METHOD setLength
  VAR
    i : UINT;
  END_VAR
                  FOR i:=0 TO cBufferSize DO
	IF (lBuffer[i] = 0) THEN
		lLength := i;
		
		IF (i>0) THEN
			lCharacters := lLength - 1;
		ELSE
			lCharacters := 0;			
		END_IF
		
		RETURN;
	END_IF
END_FOR
                
END_METHOD

METHOD appendPair
  VAR_INPUT
    parameter : STRING;
    value : STRING;
    quoted : BOOL;
    comma : BOOL;
  END_VAR
  VAR
    stmp : STRING;
  END_VAR
                  IF (comma) THEN
	stmp := CONCAT(', "',parameter);
ELSE
	stmp := CONCAT('"',parameter);
END_IF

IF (quoted) THEN
	stmp := CONCAT(stmp,'":"');
	stmp := CONCAT(stmp,value);
	stmp := CONCAT(stmp,'"');	
ELSE
	stmp := CONCAT(stmp,'":');
	stmp := CONCAT(stmp,value);
END_IF

append(stmp);
                
END_METHOD

METHOD recordTerminatorWithNewline
                  recordTerminator();
newline();
                
END_METHOD

PROPERTY Buffer : POINTER TO BYTE
GET
                    Buffer := ADR(lBuffer[0]);
                  
END_GET
END_PROPERTY

PROPERTY CurrentToken : t_parse_token_type
GET
                    CurrentToken := lCurrentToken;
                  
END_GET
END_PROPERTY

PROPERTY Length : UINT
GET
                    Length := lLength;
                  
END_GET
SET
                    lLength := Length;
checkTermination();

                  
END_SET
END_PROPERTY

PROPERTY Overflow : BOOL
GET
                    Overflow := lOverflow;
                  
END_GET
END_PROPERTY

PROPERTY NewlineStr : t_short_string
GET
                    NewlineStr := lNewline;
                  
END_GET
SET
                    lNewline := NewlineStr;
                  
END_SET
END_PROPERTY

PROPERTY Characters : UINT
GET
                    Characters := lCharacters;
                  
END_GET
END_PROPERTY

PROPERTY RecordInitiatorStr : t_short_string
GET
                    RecordInitiatorStr := lRecordInitiator;
                  
END_GET
SET
                    lRecordInitiator := RecordInitiatorStr;
                  
END_SET
END_PROPERTY

PROPERTY IndentStr : t_short_string
GET
                    IndentStr := lIndentStr;
                  
END_GET
SET
                    lIndentStr := IndentStr;
                  
END_SET
END_PROPERTY

PROPERTY RecordTerminatorStr : t_short_string
GET
                    RecordTerminatorStr := lRecordTerminator;
                  
END_GET
SET
                    lRecordTerminator := RecordTerminatorStr;
                  
END_SET
END_PROPERTY

PROPERTY BufferSize : UINT
GET
                    BufferSize := cBufferSize + 1;
                  
END_GET
END_PROPERTY
END_FUNCTION_BLOCK

FUNCTION_BLOCK StringStorex EXTENDS PersistentValue
  VAR CONSTANT
    cBufferSize : UINT := 24000;
  END_VAR
  VAR
    lValue : ARRAY[0..cBufferSize] OF BYTE;
    lLength : UINT := 0;
  END_VAR

            
          

METHOD initialize
                  lData := ADR(lValue[0]);
lCount := SIZEOF(lValue);

SUPER^.initialize();


                
END_METHOD

METHOD append
                  
                
END_METHOD

METHOD clear
                  lLength := 0;
lValue[0] := 0;
                
END_METHOD
END_FUNCTION_BLOCK

FUNCTION allocateLongString : REFERENCE TO t_long_string
  VAR_INPUT
    target : REFERENCE TO t_long_string;
  END_VAR
  VAR
    ptr : POINTER TO t_long_string;
  END_VAR

            IF (__ISVALIDREF(target)) THEN
	allocateLongString REF= target;
	RETURN;
END_IF

ptr := __NEW(t_long_string);
_countLongString := _countLongString + 1;

IF (ptr=0) THEN
	gCodeErrorHandler(pMessage:='Memory allocation failed for <t_my_string>');
	allocateLongString REF= _defaultLongString;
	RETURN;
END_IF

ptr^ := concat('allocated:',UINT_TO_STRING(_countLongString));
allocateLongString REF= ptr^;

          
END_FUNCTION

FUNCTION defineOption_1
  VAR_INPUT
    option : INT;
    token : t_token_string;
    description : t_medium_string;
  END_VAR
  VAR
    ptrptr : POINTER TO POINTER TO t_enum_option_definition;
    ptr : POINTER TO t_enum_option_definition;
    index : USINT;
    lFailed : BOOL;
    lEnumOptionMax : USINT;
  END_VAR

            index := INT_TO_USINT(option);

IF ((index>lEnumOptionMax) OR
	(ptrptr=0)) THEN
	lFailed := TRUE;
	RETURN;
END_IF

IF (ptrptr[index]=0) THEN
	gCodeErrorHandler(pMessage:='EnumRegister option already registered - check for duplicates');
	lFailed := TRUE;
	RETURN;
END_IF

ptr := __NEW(t_enum_option_definition);

IF (ptr=0) THEN
	gCodeErrorHandler(pMessage:='Memory allocation failed for enum option in <TypeHandlerEnum>');
	lFailed := TRUE;
	RETURN;
END_IF

ptrptr[index] := ptr;

ptrptr[index]^.option := option;
ptrptr[index]^.token := token;
ptrptr[index]^.description := description;
          
END_FUNCTION

FUNCTION_BLOCK TypeHandlerEnumActiveState EXTENDS TypeHandlerEnum

            
          

METHOD initialize
                  defineOption(cActiveStateNone,'none','');
defineOption(cActiveStatePre,'pre','');
defineOption(cActiveStatePost,'post','');
defineOption(cActiveStateActive,'active','');

                
END_METHOD

METHOD FB_Init : BOOL
  VAR_INPUT
    bInitRetains : BOOL;
    bInCopyCode : BOOL;
  END_VAR
                  lDefinition.option := cEnumTypeActiveState;
lDefinition.token := 'active_state';
lDefinition.description := 'States in the Active state machine';

                
END_METHOD
END_FUNCTION_BLOCK

FUNCTION_BLOCK TypeHandlerEnumBMSChargeState EXTENDS TypeHandlerEnum

            
          

METHOD initialize
                  IF ((lInitialized) OR
	(lFailed)) THEN
	RETURN;
END_IF

lEnumOptions := __NEW(ARRAY[0..cBMSChargeStateOther] OF POINTER TO t_enum_option_definition);

IF (lEnumOptions=0) THEN
	gCodeErrorHandler(pMessage:='Memory allocation failed for <TypeHandlerEnum>');
	lFailed := TRUE;
	RETURN;
END_IF

lEnumOptionMax := INT_TO_USINT(cBMSChargeStateOther);

defineOption(cBMSChargeStateShutdown,'shutdown','');
defineOption(cBMSChargeStateDC,'dc','');
defineOption(cBMSChargeStateAC,'ac','');
defineOption(cBMSChargeStateOther,'other','');

IF (NOT(lFailed)) THEN
	lInitialized := TRUE;
END_IF

                
END_METHOD

METHOD FB_Init : BOOL
  VAR_INPUT
    bInitRetains : BOOL;
    bInCopyCode : BOOL;
  END_VAR
                  lDefinition.option := cEnumTypeBMSChargeState;
lDefinition.token := 'bms_charge_state';
lDefinition.description := 'States in the BMS charge state machine';

                
END_METHOD
END_FUNCTION_BLOCK

FUNCTION_BLOCK TypeHandlerEnumBMSFaultLevel EXTENDS TypeHandlerEnum

            
          

METHOD initialize
                  IF ((lInitialized) OR
	(lFailed)) THEN
	RETURN;
END_IF

lEnumOptions := __NEW(ARRAY[0..cBMSFaultLevelSevere] OF POINTER TO t_enum_option_definition);

IF (lEnumOptions=0) THEN
	gCodeErrorHandler(pMessage:='Memory allocation failed for <TypeHandlerEnum>');
	lFailed := TRUE;
	RETURN;
END_IF

lEnumOptionMax := INT_TO_USINT(cBMSFaultLevelSevere);

defineOption(cBMSFaultLevelNone,'none','');
defineOption(cBMSFaultLevelLow,'low','');
defineOption(cBMSFaultLevelMedium,'medium','');
defineOption(cBMSFaultLevelSevere,'severe','');

IF (NOT(lFailed)) THEN
	lInitialized := TRUE;
END_IF

                
END_METHOD

METHOD FB_Init : BOOL
  VAR_INPUT
    bInitRetains : BOOL;
    bInCopyCode : BOOL;
  END_VAR
                  lDefinition.option := cEnumTypeBMSFaultLevel;
lDefinition.token := 'bms_fault_level';
lDefinition.description := 'BMS fault level';

                
END_METHOD
END_FUNCTION_BLOCK

FUNCTION_BLOCK TypeHandlerEnumBMSState EXTENDS TypeHandlerEnum

            
          

METHOD initialize
                  IF ((lInitialized) OR
	(lFailed)) THEN
	RETURN;
END_IF

lEnumOptions := __NEW(ARRAY[0..cBMSStateConnected] OF POINTER TO t_enum_option_definition);

IF (lEnumOptions=0) THEN
	gCodeErrorHandler(pMessage:='Memory allocation failed for <TypeHandlerEnum>');
	lFailed := TRUE;
	RETURN;
END_IF

lEnumOptionMax := INT_TO_USINT(cBMSStateConnected);

defineOption(cBMSStateShutdown,'shutdown','');
defineOption(cBMSStateStandby,'standby','');
defineOption(cBMSStateDisconnected,'disconnected','');
defineOption(cBMSStateConnected,'connected','');

IF (NOT(lFailed)) THEN
	lInitialized := TRUE;
END_IF

                
END_METHOD

METHOD FB_Init : BOOL
  VAR_INPUT
    bInitRetains : BOOL;
    bInCopyCode : BOOL;
  END_VAR
                  lDefinition.option := cEnumTypeBMSState;
lDefinition.token := 'bms_state';
lDefinition.description := 'States in the BMS state machine';

                
END_METHOD
END_FUNCTION_BLOCK

FUNCTION_BLOCK TypeHandlerEnumChannelMask EXTENDS TypeHandlerEnum

            
          

METHOD initialize
                  IF ((lInitialized) OR
	(lFailed)) THEN
	RETURN;
END_IF

lEnumOptions := __NEW(ARRAY[0..9] OF POINTER TO t_enum_option_definition);

IF (lEnumOptions=0) THEN
	gCodeErrorHandler(pMessage:='Memory allocation failed for <TypeHandlerEnum>');
	lFailed := TRUE;
	RETURN;
END_IF

lEnumOptionMax := INT_TO_USINT(mapping(cChannelEdgeTrace));

defineOption(cChannelNone,'none','');
defineOption(cChannelUIRadio,'Radio','');
defineOption(cChannelUICabin,'Cabin','');
defineOption(cChannelLogTCP,'Log','');
defineOption(cChannelUIRCache,'UIRCache','');
defineOption(cChannelMaster,'Master','');
defineOption(cChannelEdgeLog,'EdgeLog','');
defineOption(cChannelEdgeStateMetric,'EdgeStateMetric','');
defineOption(cChannelEdgeValueMetric,'EdgeValueMetric','');
defineOption(cChannelEdgeTrace,'EdgeTrace','');
	
IF (NOT(lFailed)) THEN
	lInitialized := TRUE;
END_IF

                
END_METHOD

METHOD FB_Init : BOOL
  VAR_INPUT
    bInitRetains : BOOL;
    bInCopyCode : BOOL;
  END_VAR
                  lDefinition.option := cEnumTypeChannelMask;
lDefinition.token := 'channel_id';
lDefinition.description := 'Channel identifiers (mask)';


                
END_METHOD

METHOD mapping : USINT
  VAR_INPUT
    option : INT;
  END_VAR
                  mapping := 0;

CASE option OF
	cChannelNone:
		mapping := 0;

	cChannelUIRadio:
		mapping := 1;

	cChannelUICabin:
		mapping := 2;

	cChannelLogTCP:
		mapping := 3;

	cChannelUIRCache:
		mapping := 4;

	cChannelMaster:
		mapping := 5;
		
	cChannelEdgeLog:
		mapping := 6;

	cChannelEdgeStateMetric:
		mapping := 7;

	cChannelEdgeValueMetric:
		mapping := 8;

	cChannelEdgeTrace:
		mapping := 9;
END_CASE
	
                
END_METHOD
END_FUNCTION_BLOCK

FUNCTION_BLOCK TypeHandlerEnumChargeQualifier EXTENDS TypeHandlerEnum

            
          

METHOD initialize
                  IF ((lInitialized) OR
	(lFailed)) THEN
	RETURN;
END_IF

lEnumOptions := __NEW(ARRAY[0..cChargeQualifierNone] OF POINTER TO t_enum_option_definition);

IF (lEnumOptions=0) THEN
	gCodeErrorHandler(pMessage:='Memory allocation failed for <TypeHandlerEnum>');
	lFailed := TRUE;
	RETURN;
END_IF

lEnumOptionMax := INT_TO_USINT(cChargeQualifierNone);

defineOption(cChargeQualifierBoth,'both','');
defineOption(cChargeQualifierCharge,'charge','');
defineOption(cChargeQualifierDischarge,'discharge','');
defineOption(cChargeQualifierNone,'none','');

IF (NOT(lFailed)) THEN
	lInitialized := TRUE;
END_IF

                
END_METHOD

METHOD FB_Init : BOOL
  VAR_INPUT
    bInitRetains : BOOL;
    bInCopyCode : BOOL;
  END_VAR
                  lDefinition.option := cEnumTypeChargeQualifier;
lDefinition.token := 'charge_qualifier';
lDefinition.description := 'Charge modulation qualifier options';

                
END_METHOD
END_FUNCTION_BLOCK

FUNCTION_BLOCK TypeHandlerEnumDataType EXTENDS TypeHandlerEnum

            
          

METHOD initialize
                  IF ((lInitialized) OR
	(lFailed)) THEN
	RETURN;
END_IF

lEnumOptions := __NEW(ARRAY[0..cDataTypeBool] OF POINTER TO t_enum_option_definition);

IF (lEnumOptions=0) THEN
	gCodeErrorHandler(pMessage:='Memory allocation failed for <TypeHandlerEnum>');
	lFailed := TRUE;
	RETURN;
END_IF

lEnumOptionMax := INT_TO_USINT(cDataTypeBool);
	
defineOption(cDataTypeNone,'none','');
defineOption(cDataTypeEnum,'enum','');
defineOption(cDataTypeString,'string','');
defineOption(cDataTypeUSINT,'usint','');
defineOption(cDataTypeUINT,'uint','');
defineOption(cDataTypeULINT,'ulint','');
defineOption(cDataTypeUDINT,'udint','');
defineOption(cDataTypeINT,'int','');
defineOption(cDataTypePercentage,'percentage','');
defineOption(cDataTypeReal,'real','');
defineOption(cDataTypeDWORD,'dword','');
defineOption(cDataTypeBool,'bool','');

IF (NOT(lFailed)) THEN
	lInitialized := TRUE;
END_IF

                
END_METHOD

METHOD FB_Init : BOOL
  VAR_INPUT
    bInitRetains : BOOL;
    bInCopyCode : BOOL;
  END_VAR
                  lDefinition.option := cEnumTypeDataType;
lDefinition.token := 'data_type';
lDefinition.description := 'Native data types';

                
END_METHOD
END_FUNCTION_BLOCK

FUNCTION_BLOCK TypeHandlerEnumDebugMask EXTENDS TypeHandlerEnum

            
          

METHOD initialize
                  IF ((lInitialized) OR
	(lFailed)) THEN
	RETURN;
END_IF

lEnumOptions := __NEW(ARRAY[0..7] OF POINTER TO t_enum_option_definition);

IF (lEnumOptions=0) THEN
	gCodeErrorHandler(pMessage:='Memory allocation failed for <TypeHandlerEnum>');
	lFailed := TRUE;
	RETURN;
END_IF

lEnumOptionMax := INT_TO_USINT(mapping(cDebugSimulateC));

defineOption(cDebugNone,'none','');
defineOption(cDebugWaitForLog,'wait_for_log','');
defineOption(cDebugEnableFailSafeOnCrash,'enbl_fail_safe','');
defineOption(cDebugDisableWatchdog,'dsbl_watch_dog','');
defineOption(cDebugSimulateCrash,'simulate_crash','');
defineOption(cDebugSimulateA,'simulate_a','');
defineOption(cDebugSimulateB,'simulate_b','');
defineOption(cDebugSimulateC,'simulate_c','');

IF (NOT(lFailed)) THEN
	lInitialized := TRUE;
END_IF

                
END_METHOD

METHOD FB_Init : BOOL
  VAR_INPUT
    bInitRetains : BOOL;
    bInCopyCode : BOOL;
  END_VAR
                  lDefinition.option := cEnumTypeDebugMask;
lDefinition.token := 'debug_flag';
lDefinition.description := 'Debug flag (mask)';

                
END_METHOD

METHOD mapping : USINT
  VAR_INPUT
    option : INT;
  END_VAR
                  mapping := 0;

CASE option OF
	cDebugNone:
		mapping := 0;

	cDebugWaitForLog:
		mapping := 1;

	cDebugEnableFailSafeOnCrash:
		mapping := 2;

	cDebugDisableWatchdog:
		mapping := 3;

	cDebugSimulateCrash:
		mapping := 4;

	cDebugSimulateA:
		mapping := 5;

	cDebugSimulateB:
		mapping := 6;

	cDebugSimulateC:
		mapping := 7;
END_CASE

	
                
END_METHOD
END_FUNCTION_BLOCK

FUNCTION_BLOCK TypeHandlerEnumExecuteReturn EXTENDS TypeHandlerEnum

            
          

METHOD initialize
                  IF ((lInitialized) OR
	(lFailed)) THEN
	RETURN;
END_IF

lEnumOptions := __NEW(ARRAY[0..cExecuteReturnReadOnly] OF POINTER TO t_enum_option_definition);

IF (lEnumOptions=0) THEN
	gCodeErrorHandler(pMessage:='Memory allocation failed for <TypeHandlerEnum>');
	lFailed := TRUE;
	RETURN;
END_IF

lEnumOptionMax := INT_TO_USINT(cExecuteReturnReadOnly);

defineOption(cExecuteReturnOK,'OK','');
defineOption(cExecuteReturnUnknownArgumentValue,'bad_arg_value','');
defineOption(cExecuteReturnUnsupportedForParticleType,'bad_for_context','');
defineOption(cExecuteReturnNullParticle,'null_object','');
defineOption(cExecuteReturnSetOverflow,'set_overflow','');
defineOption(cExecuteReturnUnknownOption,'bad_option','');	
defineOption(cExecuteReturnOKNOK,'returned_NOK','');
defineOption(cExecuteReturnUnknownCommand,'bad_command','');
defineOption(cExecuteReturnUnknownParameter,'bad_parameter','');
defineOption(cExecuteReturnUnsupportedRecurse,'illegal_recurse','');
defineOption(cExecuteReturnExecutionQueueOverflow,'queue_overflow','');
defineOption(cExecuteReturnExecutionQueueNullParticle,'null_queue_obj','');
defineOption(cExecuteReturnParseParameterError,'parameter_syntax','');
defineOption(cExecuteReturnUnknownOptionChannelMask,'bad_channel','');
defineOption(cExecuteReturnUnknownOptionDebugMask,'bad_debug_flag','');
defineOption(cExecuteReturnIllegalIndex,'illegal_index','');
defineOption(cExecuteReturnMissingArgument,'missing_arg','');
defineOption(cExecuteReturnTooFewArguments,'missing_args','');
defineOption(cExecuteReturnTooManyArguments,'extra_args','');
defineOption(cExecuteReturnInternalError,'internal','');
defineOption(cExecuteReturnPersistFailed,'persist_failed','');
defineOption(cExecuteReturnUnprocessedArguments,'unproc_args','');
defineOption(cExecuteReturnExecutionExecutorFailed,'monitor_failed','');
defineOption(cExecuteReturnExecutionSyntax,'syntax_error','');
defineOption(cExecuteReturnReadOnly,'read_only','');

IF (NOT(lFailed)) THEN
	lInitialized := TRUE;
END_IF

                
END_METHOD

METHOD FB_Init : BOOL
  VAR_INPUT
    bInitRetains : BOOL;
    bInCopyCode : BOOL;
  END_VAR
                  lDefinition.option := cEnumTypeExecuteReturn;
lDefinition.token := 'execute_return';
lDefinition.description := 'Execution exit codes';

                
END_METHOD
END_FUNCTION_BLOCK

FUNCTION_BLOCK TypeHandlerEnumFunctionalMode EXTENDS TypeHandlerEnum

            
          

METHOD initialize
                  IF ((lInitialized) OR
	(lFailed)) THEN
	RETURN;
END_IF

lEnumOptions := __NEW(ARRAY[0..cFunctionalModeTopbeamConfiguration] OF POINTER TO t_enum_option_definition);

IF (lEnumOptions=0) THEN
	gCodeErrorHandler(pMessage:='Memory allocation failed for <TypeHandlerEnum>');
	lFailed := TRUE;
	RETURN;
END_IF

lEnumOptionMax := INT_TO_USINT(cFunctionalModeTopbeamConfiguration);

defineOption(cFunctionalModeAny,'any','');
defineOption(cFunctionalModeDefault,'default','');
defineOption(cFunctionalModeTravel,'travel','');
defineOption(cFunctionalModeLift,'lift','');
defineOption(cFunctionalModeSpreaderConfiguration,'sprd_cnfg','');
defineOption(cFunctionalModeTopbeamConfiguration,'topbm_cnfg','');

IF (NOT(lFailed)) THEN
	lInitialized := TRUE;
END_IF

                
END_METHOD

METHOD FB_Init : BOOL
  VAR_INPUT
    bInitRetains : BOOL;
    bInCopyCode : BOOL;
  END_VAR
                  lDefinition.option := cEnumTypeFunctionalMode;
lDefinition.token := 'functional_mode';
lDefinition.description := 'Machine functional mode';

                
END_METHOD
END_FUNCTION_BLOCK

FUNCTION_BLOCK TypeHandlerEnumInputMode EXTENDS TypeHandlerEnum

            
          

METHOD initialize
                  IF ((lInitialized) OR
	(lFailed)) THEN
	RETURN;
END_IF

lEnumOptions := __NEW(ARRAY[0..cInputModeTopbeamConfiguration] OF POINTER TO t_enum_option_definition);

IF (lEnumOptions=0) THEN
	gCodeErrorHandler(pMessage:='Memory allocation failed for <TypeHandlerEnum>');
	lFailed := TRUE;
	RETURN;
END_IF

lEnumOptionMax := INT_TO_USINT(cInputModeTopbeamConfiguration);

defineOption(cInputModeNone,'none','');
defineOption(cInputModeDefault,'default','');
defineOption(cInputModeSpreaderConfiguration,'sprd_cnfg','');
defineOption(cInputModeTopbeamConfiguration,'topbm_cnfg','');

IF (NOT(lFailed)) THEN
	lInitialized := TRUE;
END_IF

                
END_METHOD

METHOD FB_Init : BOOL
  VAR_INPUT
    bInitRetains : BOOL;
    bInCopyCode : BOOL;
  END_VAR
                  lDefinition.option := cEnumTypeInputMode;
lDefinition.token := 'input_mode';
lDefinition.description := 'Machine input mode';

                
END_METHOD
END_FUNCTION_BLOCK

FUNCTION_BLOCK TypeHandlerEnumLockState EXTENDS TypeHandlerEnum

            
          

METHOD initialize
                  IF ((lInitialized) OR
	(lFailed)) THEN
	RETURN;
END_IF

lEnumOptions := __NEW(ARRAY[0..cLockStatePartial] OF POINTER TO t_enum_option_definition);

IF (lEnumOptions=0) THEN
	gCodeErrorHandler(pMessage:='Memory allocation failed for <TypeHandlerEnum>');
	lFailed := TRUE;
	RETURN;
END_IF

lEnumOptionMax := INT_TO_USINT(cLockStatePartial);

defineOption(cLockStateNone,'none','');
defineOption(cLockStateUnlocked,'unlocked','');
defineOption(cLockStateLocked,'locked','');
defineOption(cLockStatePartial,'partial','');

IF (NOT(lFailed)) THEN
	lInitialized := TRUE;
END_IF

                
END_METHOD

METHOD FB_Init : BOOL
  VAR_INPUT
    bInitRetains : BOOL;
    bInCopyCode : BOOL;
  END_VAR
                  lDefinition.option := cEnumTypeLockState;
lDefinition.token := 'lock_state';
lDefinition.description := 'Twistlock lock state';

                
END_METHOD
END_FUNCTION_BLOCK

FUNCTION_BLOCK TypeHandlerEnumOBCState EXTENDS TypeHandlerEnum

            
          

METHOD initialize
                  IF ((lInitialized) OR
	(lFailed)) THEN
	RETURN;
END_IF

lEnumOptions := __NEW(ARRAY[0..cOBCStateError] OF POINTER TO t_enum_option_definition);

IF (lEnumOptions=0) THEN
	gCodeErrorHandler(pMessage:='Memory allocation failed for <TypeHandlerEnum>');
	lFailed := TRUE;
	RETURN;
END_IF

lEnumOptionMax := INT_TO_USINT(cOBCStateError);

defineOption(cOBCStateDisconnected,'disconnect','');
defineOption(cOBCStateCharging,'charging','');
defineOption(cOBCStateStandby,'standby','');
defineOption(cOBCStateError,'error','');

IF (NOT(lFailed)) THEN
	lInitialized := TRUE;
END_IF

                
END_METHOD

METHOD FB_Init : BOOL
  VAR_INPUT
    bInitRetains : BOOL;
    bInCopyCode : BOOL;
  END_VAR
                  lDefinition.option := cEnumTypeOBCState;
lDefinition.token := 'obc_state';
lDefinition.description := 'Onboard charger state';

                
END_METHOD
END_FUNCTION_BLOCK

FUNCTION_BLOCK TypeHandlerEnumOBCStatus EXTENDS TypeHandlerEnum

            
          

METHOD initialize
                  IF ((lInitialized) OR
	(lFailed)) THEN
	RETURN;
END_IF

lEnumOptions := __NEW(ARRAY[0..cOBCStatusError] OF POINTER TO t_enum_option_definition);

IF (lEnumOptions=0) THEN
	gCodeErrorHandler(pMessage:='Memory allocation failed for <TypeHandlerEnum>');
	lFailed := TRUE;
	RETURN;
END_IF

lEnumOptionMax := INT_TO_USINT(cOBCStatusError);

defineOption(cOBCStatusNone,'none','');
defineOption(cOBCStatusCharging,'charging','');
defineOption(cOBCStatusStandby,'standby','');
defineOption(cOBCStatusError,'error','');

IF (NOT(lFailed)) THEN
	lInitialized := TRUE;
END_IF

                
END_METHOD

METHOD FB_Init : BOOL
  VAR_INPUT
    bInitRetains : BOOL;
    bInCopyCode : BOOL;
  END_VAR
                  lDefinition.option := cEnumTypeOBCStatus;
lDefinition.token := 'obc_status';
lDefinition.description := 'Onboard charger status';

                
END_METHOD
END_FUNCTION_BLOCK

FUNCTION_BLOCK TypeHandlerEnumOperatingMethod EXTENDS TypeHandlerEnum

            
          

METHOD initialize
                  IF ((lInitialized) OR
	(lFailed)) THEN
	RETURN;
END_IF

lEnumOptions := __NEW(ARRAY[0..cOperatingMethodNormal] OF POINTER TO t_enum_option_definition);

IF (lEnumOptions=0) THEN
	gCodeErrorHandler(pMessage:='Memory allocation failed for <TypeHandlerEnum>');
	lFailed := TRUE;
	RETURN;
END_IF

lEnumOptionMax := INT_TO_USINT(cOperatingMethodNormal);

defineOption(cOperatingMethodNone,'none','');
defineOption(cOperatingMethodPark,'park','');
defineOption(cOperatingMethodUnpark,'unpark','');
defineOption(cOperatingMethodLock,'lock','');
defineOption(cOperatingMethodLockWithoutPark,'lock_no_park','');
defineOption(cOperatingMethodUnlock,'unlock','');
defineOption(cOperatingMethodSlow,'slow','');
defineOption(cOperatingMethodNormal,'normal','');

IF (NOT(lFailed)) THEN
	lInitialized := TRUE;
END_IF

                
END_METHOD

METHOD FB_Init : BOOL
  VAR_INPUT
    bInitRetains : BOOL;
    bInCopyCode : BOOL;
  END_VAR
                  lDefinition.option := cEnumTypeOperatingMethod;
lDefinition.token := 'operating_method';
lDefinition.description := 'Operating mode commands';

                
END_METHOD
END_FUNCTION_BLOCK

FUNCTION_BLOCK TypeHandlerEnumProgMovCode EXTENDS TypeHandlerEnum

            
          

METHOD initialize
                  IF ((lInitialized) OR
	(lFailed)) THEN
	RETURN;
END_IF

lEnumOptions := __NEW(ARRAY[0..cOBCStatusError] OF POINTER TO t_enum_option_definition);

IF (lEnumOptions=0) THEN
	gCodeErrorHandler(pMessage:='Memory allocation failed for <TypeHandlerEnum>');
	lFailed := TRUE;
	RETURN;
END_IF

lEnumOptionMax := INT_TO_USINT(cOBCStatusError);

defineOption(cProgMovCodeNone,'none','');
defineOption(cProgMovCode_Steer_0,'steer_0','');
	
IF (NOT(lFailed)) THEN
	lInitialized := TRUE;
END_IF

                
END_METHOD

METHOD FB_Init : BOOL
  VAR_INPUT
    bInitRetains : BOOL;
    bInCopyCode : BOOL;
  END_VAR
                  lDefinition.option := cEnumTypeProgMovCode;
lDefinition.token := 'progmov_code';
lDefinition.description := 'Automation code';

                
END_METHOD
END_FUNCTION_BLOCK

FUNCTION_BLOCK TypeHandlerEnumRunState EXTENDS TypeHandlerEnum

            
          

METHOD initialize
                  IF ((lInitialized) OR
	(lFailed)) THEN
	RETURN;
END_IF

lEnumOptions := __NEW(ARRAY[0..cRunStateStop] OF POINTER TO t_enum_option_definition);

IF (lEnumOptions=0) THEN
	gCodeErrorHandler(pMessage:='Memory allocation failed for <TypeHandlerEnum>');
	lFailed := TRUE;
	RETURN;
END_IF

lEnumOptionMax := INT_TO_USINT(cRunStateStop);

defineOption(cRunStateNone,'none','');
defineOption(cRunStateStart,'start','');
defineOption(cRunStateStop,'stop','');

IF (NOT(lFailed)) THEN
	lInitialized := TRUE;
END_IF

                
END_METHOD

METHOD FB_Init : BOOL
  VAR_INPUT
    bInitRetains : BOOL;
    bInCopyCode : BOOL;
  END_VAR
                  lDefinition.option := cEnumTypeRunState;
lDefinition.token := 'run_state';
lDefinition.description := 'Run state machine';

                
END_METHOD
END_FUNCTION_BLOCK

FUNCTION_BLOCK TypeHandlerEnumSeverity EXTENDS TypeHandlerEnum

            
          

METHOD initialize
                  IF ((lInitialized) OR
	(lFailed)) THEN
	RETURN;
END_IF

lEnumOptions := __NEW(ARRAY[0..cSeverityCritical] OF POINTER TO t_enum_option_definition);

IF (lEnumOptions=0) THEN
	gCodeErrorHandler(pMessage:='Memory allocation failed for <TypeHandlerEnum>');
	lFailed := TRUE;
	RETURN;
END_IF

lEnumOptionMax := INT_TO_USINT(cSeverityCritical);

defineOption(cSeverityNone,'none','');
defineOption(cSeverityWarning,'warning','');
defineOption(cSeverityError,'error','');
defineOption(cSeverityCritical,'critical','');

IF (NOT(lFailed)) THEN
	lInitialized := TRUE;
END_IF

                
END_METHOD

METHOD FB_Init : BOOL
  VAR_INPUT
    bInitRetains : BOOL;
    bInCopyCode : BOOL;
  END_VAR
                  lDefinition.option := cEnumTypeSeverity;
lDefinition.token := 'severity';
lDefinition.description := 'Severity options';

                
END_METHOD
END_FUNCTION_BLOCK

FUNCTION_BLOCK TypeHandlerEnumShutdownCode EXTENDS TypeHandlerEnum

            
          

METHOD initialize
                  IF ((lInitialized) OR
	(lFailed)) THEN
	RETURN;
END_IF

lEnumOptions := __NEW(ARRAY[0..cShutdownCodeTrapDetected] OF POINTER TO t_enum_option_definition);

IF (lEnumOptions=0) THEN
	gCodeErrorHandler(pMessage:='Memory allocation failed for <TypeHandlerEnum>');
	lFailed := TRUE;
	RETURN;
END_IF

lEnumOptionMax := INT_TO_USINT(cShutdownCodeTrapDetected);

defineOption(cShutdownCodeUnknown,'unknown','');
defineOption(cShutdownCodeIgnition,'ignition','');
defineOption(cShutdownCodeSoftware,'software','');
defineOption(cShutdownCodeSupervisor,'supervisor','');
defineOption(cShutdownCodeCrashDetected,'crash','');
defineOption(cShutdownCodeTrapDetected,'trap','');

IF (NOT(lFailed)) THEN
	lInitialized := TRUE;
END_IF

                
END_METHOD

METHOD FB_Init : BOOL
  VAR_INPUT
    bInitRetains : BOOL;
    bInCopyCode : BOOL;
  END_VAR
                  lDefinition.option := cEnumTypeShutdownCode;
lDefinition.token := 'shutdown_code';
lDefinition.description := 'Device shutdown diagnostic';

                
END_METHOD
END_FUNCTION_BLOCK

FUNCTION_BLOCK TypeHandlerEnumSteerMode EXTENDS TypeHandlerEnum

            
          

METHOD initialize
                  IF ((lInitialized) OR
	(lFailed)) THEN
	RETURN;
END_IF

lEnumOptions := __NEW(ARRAY[0..cSteerModeCustom] OF POINTER TO t_enum_option_definition);

IF (lEnumOptions=0) THEN
	gCodeErrorHandler(pMessage:='Memory allocation failed for <TypeHandlerEnum>');
	lFailed := TRUE;
	RETURN;
END_IF

lEnumOptionMax := INT_TO_USINT(cSteerModeCustom);

defineOption(cSteerModeNone,'none','');
defineOption(cSteerMode4WS,'4ws','');
defineOption(cSteerModeLateral,'lateral','');
defineOption(cSteerModeCarousel,'carousel','');
defineOption(cSteerModeReconfigure,'reconfigure','');
defineOption(cSteerModeLateralNeg90,'lat_neg_90','');
defineOption(cSteerModeLateralPos90,'lat_pos_90','');
defineOption(cSteerModeCustom,'custom','');

IF (NOT(lFailed)) THEN
	lInitialized := TRUE;
END_IF

                
END_METHOD

METHOD FB_Init : BOOL
  VAR_INPUT
    bInitRetains : BOOL;
    bInCopyCode : BOOL;
  END_VAR
                  lDefinition.option := cEnumTypeSteerMode;
lDefinition.token := 'steer_mode';
lDefinition.description := 'Steering modes';

                
END_METHOD
END_FUNCTION_BLOCK

FUNCTION_BLOCK TypeHandlerEnumSubsystem EXTENDS TypeHandlerEnum

            
          

METHOD initialize
                  IF ((lInitialized) OR
	(lFailed)) THEN
	RETURN;
END_IF

lEnumOptions := __NEW(ARRAY[0..cSubsystemMachine] OF POINTER TO t_enum_option_definition);

IF (lEnumOptions=0) THEN
	gCodeErrorHandler(pMessage:='Memory allocation failed for <TypeHandlerEnum>');
	lFailed := TRUE;
	RETURN;
END_IF

lEnumOptionMax := INT_TO_USINT(cSubsystemMachine);

defineOption(cSubsystemNone,'none','');
defineOption(cSubsystemSpreader,'Spreader','');
defineOption(cSubsystemBeacons,'Beacons','');
defineOption(cSubsystemCabin,'Cabin','');
defineOption(cSubsystemLights,'Lights','');
defineOption(cSubsystemPowerpack,'owerpack','');
defineOption(cSubsystemSideshiftAB,'SideshiftAB','');
defineOption(cSubsystemSideshiftCD,'SideshiftCD','');
defineOption(cSubsystemSpreaderPowerPack,'SprPowerPack','');
defineOption(cSubsystemSteerA,'SteerA','');
defineOption(cSubsystemSteerB,'SteerB','');
defineOption(cSubsystemSteerC,'SteerC','');
defineOption(cSubsystemSteerD,'SteerD','');
defineOption(cSubsystemTravelA,'TravelA','');
defineOption(cSubsystemTravelB,'TravelB','');
defineOption(cSubsystemTravelC,'TravelC','');
defineOption(cSubsystemTravelD,'TravelD','');
defineOption(cSubsystemWinchA,'WinchA','');
defineOption(cSubsystemWinchB,'WinchB','');
defineOption(cSubsystemWinchC,'WinchC','');
defineOption(cSubsystemWinchD,'WinchD','');
defineOption(cSubsystemTwistlockA,'TwistlockA','');
defineOption(cSubsystemTwistlockB,'TwistlockB','');
defineOption(cSubsystemTwistlockC,'TwistlockC','');
defineOption(cSubsystemTwistlockD,'TwistlockD','');
defineOption(cSubsystemTopbeamAB,'TopbeamAB','');
defineOption(cSubsystemTopbeamCD,'TopbeamCD','');
defineOption(cSubsystemCANBusSystem,'CANBusSystem','');
defineOption(cSubsystemCANBusDrive,'CANBusDrive','');
defineOption(cSubsystemBattery,'Battery','');
defineOption(cSubsystemSecondary,'Secondary','');
defineOption(cSubsystemUInterface,'UInterface','');
defineOption(cSubsystemHydraulics,'Hydraulics','');
defineOption(cSubsystemLift,'Lift','');
defineOption(cSubsystemTravel,'Travel','');
defineOption(cSubsystemSteer,'Steer','');
defineOption(cSubsystemMachine,'Machine','');

IF (NOT(lFailed)) THEN
	lInitialized := TRUE;
END_IF

                
END_METHOD

METHOD FB_Init : BOOL
  VAR_INPUT
    bInitRetains : BOOL;
    bInCopyCode : BOOL;
  END_VAR
                  lDefinition.option := cEnumTypeSubsystem;
lDefinition.token := 'subsystem';
lDefinition.description := 'Machine subsystems';

                
END_METHOD
END_FUNCTION_BLOCK

FUNCTION_BLOCK TypeHandlerEnumSystemControl EXTENDS TypeHandlerEnum

            
          

METHOD initialize
                  IF ((lInitialized) OR
	(lFailed)) THEN
	RETURN;
END_IF

lEnumOptions := __NEW(ARRAY[0..cSystemControlNone] OF POINTER TO t_enum_option_definition);

IF (lEnumOptions=0) THEN
	gCodeErrorHandler(pMessage:='Memory allocation failed for <TypeHandlerEnum>');
	lFailed := TRUE;
	RETURN;
END_IF

lEnumOptionMax := INT_TO_USINT(cSystemControlNone);

defineOption(cSystemControlReset,'reset','');
defineOption(cSystemControlEStop,'estop','');
defineOption(cSystemControlStop,'stop','');
defineOption(cSystemControlStart,'start','');
defineOption(cSystemControlNone,'none','');

IF (NOT(lFailed)) THEN
	lInitialized := TRUE;
END_IF

                
END_METHOD

METHOD FB_Init : BOOL
  VAR_INPUT
    bInitRetains : BOOL;
    bInCopyCode : BOOL;
  END_VAR
                  lDefinition.option := cEnumTypeSystemControl;
lDefinition.token := 'system_control';
lDefinition.description := 'Options for controlling system state';

                
END_METHOD
END_FUNCTION_BLOCK

FUNCTION_BLOCK TypeHandlerEnumSystemState EXTENDS TypeHandlerEnum

            
          

METHOD initialize
                  IF ((lInitialized) OR
	(lFailed)) THEN
	RETURN;
END_IF

lEnumOptions := __NEW(ARRAY[0..cSystemStateOperational] OF POINTER TO t_enum_option_definition);

IF (lEnumOptions=0) THEN
	gCodeErrorHandler(pMessage:='Memory allocation failed for <TypeHandlerEnum>');
	lFailed := TRUE;
	RETURN;
END_IF

lEnumOptionMax := INT_TO_USINT(cSystemStateOperational);

defineOption(cSystemStateNone,'none','');
defineOption(cSystemStateInitialized,'initialized','');
defineOption(cSystemStateStandby,'standby','');
defineOption(cSystemStatePreparing,'preparing','');
defineOption(cSystemStateCharging,'charging','');
defineOption(cSystemStatePreOperational,'pre_operational','');
defineOption(cSystemStatePoweringDown,'powering_down','');
defineOption(cSystemStatePoweringUp,'powering_up','');
defineOption(cSystemStateGoOperational,'go_operational','');
defineOption(cSystemStateExitOperational,'exit_operational','');
defineOption(cSystemStateOperational,'operational','');

IF (NOT(lFailed)) THEN
	lInitialized := TRUE;
END_IF

                
END_METHOD

METHOD FB_Init : BOOL
  VAR_INPUT
    bInitRetains : BOOL;
    bInCopyCode : BOOL;
  END_VAR
                  lDefinition.option := cEnumTypeSystemState;
lDefinition.token := 'system_state';
lDefinition.description := 'System state machine';

                
END_METHOD
END_FUNCTION_BLOCK

FUNCTION_BLOCK TypeHandlerEnumTMSState EXTENDS TypeHandlerEnum

            
          

METHOD initialize
                  IF ((lInitialized) OR
	(lFailed)) THEN
	RETURN;
END_IF

lEnumOptions := __NEW(ARRAY[0..cTMSStateCirculation] OF POINTER TO t_enum_option_definition);

IF (lEnumOptions=0) THEN
	gCodeErrorHandler(pMessage:='Memory allocation failed for <TypeHandlerEnum>');
	lFailed := TRUE;
	RETURN;
END_IF

lEnumOptionMax := INT_TO_USINT(cTMSStateCirculation);

defineOption(cTMSStateShutdown,'shutdown','');
defineOption(cTMSStateCooling,'cooling','');
defineOption(cTMSStateHeating,'heating','');
defineOption(cTMSStateCirculation,'circulation','');

IF (NOT(lFailed)) THEN
	lInitialized := TRUE;
END_IF

                
END_METHOD

METHOD FB_Init : BOOL
  VAR_INPUT
    bInitRetains : BOOL;
    bInCopyCode : BOOL;
  END_VAR
                  lDefinition.option := cEnumTypeTMSState;
lDefinition.token := 'tms_state';
lDefinition.description := 'Battery thermal management state';

                
END_METHOD
END_FUNCTION_BLOCK

FUNCTION_BLOCK TypeHandlerEnumTokenType EXTENDS TypeHandlerEnum

            
          

METHOD initialize
                  IF ((lInitialized) OR
	(lFailed)) THEN
	RETURN;
END_IF

lEnumOptions := __NEW(ARRAY[0..cTokenImport] OF POINTER TO t_enum_option_definition);

IF (lEnumOptions=0) THEN
	gCodeErrorHandler(pMessage:='Memory allocation failed for <TypeHandlerEnum>');
	lFailed := TRUE;
	RETURN;
END_IF

lEnumOptionMax := INT_TO_USINT(cTokenImport);

defineOption(cTokenNone,'none','');
defineOption(cTokenDescribe,'describe','');
defineOption(cTokenSyntax,'syntax','');
defineOption(cTokenVerify,'verify','');
defineOption(cTokenIdentify,'identify','');
defineOption(cTokenRegister,'register','');
defineOption(cTokenConfigure,'configure','');
defineOption(cTokenSetFailSafeMode,'failsafe_set','');
defineOption(cTokenClearFailSafeMode,'failsafe_clr','');
defineOption(cTokenFailSafeConfig,'failsafe_cnfg','');
defineOption(cTokenProceed,'proceed','');
defineOption(cTokenList,'list','');
defineOption(cTokenDebugMaskAdd,'debug_add','');
defineOption(cTokenDebugMaskDelete,'debug_del','');
defineOption(cTokenDebugMaskClear,'debug_clr','');
defineOption(cTokenClose,'close','');
defineOption(cTokenExport,'export','');
defineOption(cTokenClear,'clear','');
defineOption(cTokenDeregister,'deregister','');
defineOption(cTokenTrigger,'trigger','');
defineOption(cTokenChannelMaskAdd,'chanmask_add','');
defineOption(cTokenChannelMaskDelete,'chanmask_del','');
defineOption(cTokenChannelMaskClear,'chanmask_clr','');
defineOption(cTokenChannelIndex,'channel','');
defineOption(cTokenValue,'value','');
defineOption(cTokenOverrideValue,'override_value','');
defineOption(cTokenOverride,'override','');
defineOption(cTokenValueType,'value_type','');
defineOption(cTokenMeaning,'meaning','');
defineOption(cTokenOverrideMeaning,'override_meaning','');
defineOption(cTokenRawIndex,'raw_index','');
defineOption(cTokenIndex,'index','');
defineOption(cTokenUnknown,'unknown','');
defineOption(cTokenObject,'object','');
defineOption(cTokenFeature,'arg','');
defineOption(cTokenZero,'zero','');
defineOption(sTokenUpper,'upper','');
defineOption(cTokenImport,'import','');

IF (NOT(lFailed)) THEN
	lInitialized := TRUE;
END_IF

                
END_METHOD

METHOD FB_Init : BOOL
  VAR_INPUT
    bInitRetains : BOOL;
    bInCopyCode : BOOL;
  END_VAR
                  lDefinition.option := cEnumTypeTokenType;
lDefinition.token := 'token_type';
lDefinition.description := 'Standard tokens';

                
END_METHOD
END_FUNCTION_BLOCK

FUNCTION_BLOCK TypeHandlerEnumUIEventCode EXTENDS TypeHandlerEnum

            
          

METHOD initialize
                  IF ((lInitialized) OR
	(lFailed)) THEN
	RETURN;
END_IF

lEnumOptions := __NEW(ARRAY[0..cUIEventCodeProgMovStart] OF POINTER TO t_enum_option_definition);

IF (lEnumOptions=0) THEN
	gCodeErrorHandler(pMessage:='Memory allocation failed for <TypeHandlerEnum>');
	lFailed := TRUE;
	RETURN;
END_IF

lEnumOptionMax := INT_TO_USINT(cUIEventCodeProgMovStart);

defineOption(cUIEventCodeNone,'none','');
defineOption(cUIEventCodeToggleLights,'toggle_lights','');
defineOption(cUIEventCodeUIModeResponse,'ui_mode_resp','');
defineOption(cUIEventCodeToggleSpreaderConfiguration,'sprd_cnfg','');
defineOption(cUIEventCodeSpreaderExtensionAutoCommand,'sprd_extend','');
defineOption(cUIEventCodeSpreaderRetractionAutoCommand,'sprd_retract','');
defineOption(cUIEventCodeInitiate,'initiate','');
defineOption(cUIEventCodeStart,'start','');
defineOption(cUIEventCodeStop,'stop','');
defineOption(cUIEventCodeProgMovStart,'prog_move_start','');

IF (NOT(lFailed)) THEN
	lInitialized := TRUE;
END_IF

                
END_METHOD

METHOD FB_Init : BOOL
  VAR_INPUT
    bInitRetains : BOOL;
    bInCopyCode : BOOL;
  END_VAR
                  lDefinition.option := cEnumTypeUiEventCode;
lDefinition.token := 'ui_event_code';
lDefinition.description := 'User Interface event code';

                
END_METHOD
END_FUNCTION_BLOCK

FUNCTION_BLOCK TypeHandlerEnumUIOrientation EXTENDS TypeHandlerEnum

            
          

METHOD initialize
                  IF ((lInitialized) OR
	(lFailed)) THEN
	RETURN;
END_IF

lEnumOptions := __NEW(ARRAY[0..cUIOrientationOpposite] OF POINTER TO t_enum_option_definition);

IF (lEnumOptions=0) THEN
	gCodeErrorHandler(pMessage:='Memory allocation failed for <TypeHandlerEnum>');
	lFailed := TRUE;
	RETURN;
END_IF

lEnumOptionMax := INT_TO_USINT(cUIOrientationOpposite);

defineOption(cUIOrientationNone,'none','');
defineOption(cUIOrientationForward,'forward','');
defineOption(cUIOrientationSide,'side','');
defineOption(cUIOrientationReverse,'reverse','');
defineOption(cUIOrientationOpposite,'opposite','');

IF (NOT(lFailed)) THEN
	lInitialized := TRUE;
END_IF

                
END_METHOD

METHOD FB_Init : BOOL
  VAR_INPUT
    bInitRetains : BOOL;
    bInCopyCode : BOOL;
  END_VAR
                  lDefinition.option := cEnumTypeUiOrientation;
lDefinition.token := 'ui_orientation';
lDefinition.description := 'User Interface orientation';

                
END_METHOD
END_FUNCTION_BLOCK

FUNCTION_BLOCK TypeHandlerEnumValueStyle EXTENDS TypeHandlerEnum

            
          

METHOD initialize
                  IF ((lInitialized) OR
	(lFailed)) THEN
	RETURN;
END_IF

lEnumOptions := __NEW(ARRAY[0..cValueStyleTrigger] OF POINTER TO t_enum_option_definition);

IF (lEnumOptions=0) THEN
	gCodeErrorHandler(pMessage:='Memory allocation failed for <TypeHandlerEnum>');
	lFailed := TRUE;
	RETURN;
END_IF

lEnumOptionMax := INT_TO_USINT(cValueStyleTrigger);

defineOption(cValueStyleConfigurable,'configurable','');
defineOption(cValueStyleParameter,'parameter','');
defineOption(cValueStyleTrigger,'trigger','');

IF (NOT(lFailed)) THEN
	lInitialized := TRUE;
END_IF

                
END_METHOD

METHOD FB_Init : BOOL
  VAR_INPUT
    bInitRetains : BOOL;
    bInCopyCode : BOOL;
  END_VAR
                  lDefinition.option := cEnumTypeValueStyle;
lDefinition.token := 'value_style';
lDefinition.description := 'How a value is treated';

                
END_METHOD
END_FUNCTION_BLOCK

FUNCTION getStringForEventCode : t_medium_string
  VAR_INPUT
    code : t_event_code;
  END_VAR

            getStringForEventCode := 'event';

CASE code OF
	cECNone:
		getStringForEventCode := 'none';

	cECSystemControl:
		getStringForEventCode := 'SysStateCntrl';

	cECAllowUpState:
		getStringForEventCode := 'SysStateAllowUp';

	cECAllowDownState:
		getStringForEventCode := 'SysStateAllowDn';

	cECForceMaxState:
		getStringForEventCode := 'SysStateMax';

	cECNextState:
		getStringForEventCode := 'SysStateNext';

	cECModulation:
		getStringForEventCode := 'SysStateMod';

	cECChargeModulation:
		getStringForEventCode := 'SysStateChrgMod';

	cECMovementInputInterlock:
		getStringForEventCode := 'iMovInput';

	cECMovementChargeInterlock:
		getStringForEventCode := 'iMovChrg';

	cECSecondaryPowerModulation:
		getStringForEventCode := 'SecPwrMod';

	cECTransitionInitializedStandby:
		getStringForEventCode := 'sstInitStdby';

	cECTransitionStandbyPreparing:
		getStringForEventCode := 'sstStdbyPrep';

	cECTransitionStandbyInitialized:
		getStringForEventCode := 'sstStbyInit';

	cECTransitionPreparingPreOperational:
		getStringForEventCode := 'sstPrepPreOp';

	cECTransitionPreparingCharging:
		getStringForEventCode := 'sstPrepChrg';

	cECTransitionPreparingStandby:
		getStringForEventCode := 'sstPrepStdby';

	cECTransitionChargingPreparing:
		getStringForEventCode := 'sstChrgPrep';

	cECTransitionPreOperationalPreparing:
		getStringForEventCode := 'sstPreOpPrep';

	cECTransitionPoweringUpGoOperational:
		getStringForEventCode := 'sstPwrUpGoOp';

	cECTransitionGoOperationalOperational:
		getStringForEventCode := 'sstGoOpOper';

	cECTransitionExitOperationalPoweringDown:
		getStringForEventCode := 'sstExOpPwrDn';

	cECTransitionPoweringDownPreOperational:
		getStringForEventCode := 'sstPwrDnPreOp';
		
	cECMetric:
		getStringForEventCode := 'Metric';	
END_CASE

IF (strcmp(getStringForEventCode,'event')) THEN
	gEventCodeLastUnknown := code;
END_IF
          
END_FUNCTION

FUNCTION getStringForParseTokenType : t_medium_string
  VAR_INPUT
    token : t_parse_token_type;
  END_VAR

            getStringForParseTokenType := 'none';		

CASE token OF
	cParseTokenOverflow:
		getStringForParseTokenType := 'overflow';
		
	cParseTokenError:
		getStringForParseTokenType := 'error';

	cParseTokenSimple:
		getStringForParseTokenType := 'command';
		
	cParseTokenName:
		getStringForParseTokenType := 'name';
		
	cParseTokenParameter:
		getStringForParseTokenType := 'parameter';
		
	cParseTokenOption:
		getStringForParseTokenType := 'option';
	
	cParseTokenTerminator:
		getStringForParseTokenType := 'terminator';
		
	cParseTokenFinished:
		getStringForParseTokenType := 'finished';
END_CASE
          
END_FUNCTION

FUNCTION getStringForStateCode : t_medium_string
  VAR_INPUT
    code : t_state_code;
  END_VAR

            getStringForStateCode :='state';

CASE code OF
	cSCNone:
		getStringForStateCode := 'none';

	cACSteerALargeSensorDelta:
		getStringForStateCode := 'LrgSensorDelta';

	cACSecondaryNotRunning:
		getStringForStateCode := 'SecPwrNotRun';

	cACSecondaryNotRunningModulation:
		getStringForStateCode := 'SecPwrNotRunMod';

	cACSecondaryWaiting:
		getStringForStateCode := 'SecPwrWait';

	cACSecondaryRunStateMismatch:
		getStringForStateCode := 'SecPwrMismatch';

	cACSecondaryTemperature:
		getStringForStateCode := 'SecPwrTemp';
	
	cACChannelNotGood:
		getStringForStateCode := 'MasterNotGood';

	cACChannelOperationalFail:
		getStringForStateCode := 'MasterOpFail';

	cACChannelNotOperational:
		getStringForStateCode := 'MasterNotOp';

	cACChannelOverflow:
		getStringForStateCode := 'MasterOverflow';

	cACChannelSlaveFailed:
		getStringForStateCode := 'MasterSlaveFail';

	cACCANOpenSlaveNotOperational:
		getStringForStateCode := 'SlaveNotOp';

	cACCANOpenSlaveModulation:
		getStringForStateCode := 'SlaveMod';

	cACCANOpenSlaveAllowableUp:
		getStringForStateCode := 'SlaveAllowUp';

	cACCANOpenMasterNotOperational:
		getStringForStateCode := 'MasterNotOp';

	cACCANOpenMasterModulation:
		getStringForStateCode := 'MasterMod';

	cACCANOpenMasterAllowableUp:
		getStringForStateCode := 'MasterAllowUp';
	
	cACCANOpenSlaveNoValidTransmissions:
		getStringForStateCode := 'SlaveNoVldTrnms';

	cACCANOpenSlaveNotify:
		getStringForStateCode := 'SlaveNotify';

	cACCANOpenSlaveBlock:
		getStringForStateCode := 'SlaveBlock';

	cACCANOpenSlaveStop:
		getStringForStateCode := 'SlaveStop';
		
	cACUInterfaceEstop:
		getStringForStateCode := 'UIEstop';

	cACUInterfaceStop:
		getStringForStateCode := 'UIStop';

	cACUInterfaceEmgy:
		getStringForStateCode := 'UIEmgy';

	cACUInterfaceNotReady:
		getStringForStateCode := 'UINotRdy';

	cACControllerTemperatureCutback:
		getStringForStateCode := 'CntTempCutb';
		
	cACMotorTemperatureCutback:
		getStringForStateCode := 'MotTempCutb';

	cACMotorTemperatureSensor:
		getStringForStateCode := 'MotTempSensor';

	cACCoolantReservoir:
		getStringForStateCode := 'ClntReserv';

	cACCoolantTempHotCutback:
		getStringForStateCode := 'ClntTempHotCutb';

	cACCoolantTempColdCutback:
		getStringForStateCode := 'ClntTempColdCutb';

	cACCoolantHeating:
		getStringForStateCode := 'ClntHeating';

	cACCoolantChilling:
		getStringForStateCode := 'ClntChilling';

	cACCoolantSecondaryPowerFailHeatingCooling:
		getStringForStateCode := 'ClntSecFailHC';

	cACCoolantSecondaryPowerFailPump:
		getStringForStateCode := 'ClntSecFailPmp';

	cACChargerOBCError:
		getStringForStateCode := 'ChrgOBCErr';

	cACBMSAvailabilityInsufficient:
		getStringForStateCode := 'BMSAvailInsuff';

	cACBMSAvailabilityLimited:
		getStringForStateCode := 'BMSAvailLmtd';

	cBMSChargeAvailabilityLimited:
		getStringForStateCode := 'BMSChrgAvailLm';

	cBMSChargeAvailabilityLimitedSevere:
		getStringForStateCode := 'BMSChrgAvailLmSv';

	cBMSDischargeAvailabilityLimited:
		getStringForStateCode := 'BMSDschAvailLm';

	cBMSDischargeAvailabilityLimitedSevere:
		getStringForStateCode := 'BMSDschAvailLmSv';
		
	cACBMSRequestDisconnect:
		getStringForStateCode := 'BMSReqDisconnect';
	
	cACSOCBelowOperatingMinimum:
		getStringForStateCode := 'SOCLowOpMin';

	cACSOCBelowStandbyMinimum:
		getStringForStateCode := 'SOCLowStdbyMin';

	cACSOCWarningLow:
		getStringForStateCode := 'SOCWarnLow';
	
	cACBMSNotConnected:
		getStringForStateCode := 'BMSNotConnect';
		
	cACBMSFailToConnect:
		getStringForStateCode := 'BMSNotConnect';

	cACBMSChargeCutback:
		getStringForStateCode := 'BMSChrgCutb';

	cACBMSDischargeCutback:
		getStringForStateCode := 'BMSDischCutb';

	cACBackupBatteryVoltageLow:
		getStringForStateCode := 'BckupBatVltLow';

	cACBeaconsSecondaryPowerFail:
		getStringForStateCode := 'BcnsSecPwrFail';

	cACSecondaryPowerFail:
		getStringForStateCode := 'BeepSecPwrFail';

	cACTMSStateMismatch:
		getStringForStateCode := 'TMSMismatch';

	cACBMSChargeStateMismatch:
		getStringForStateCode := 'BMSChrgMismatch';
		
	cACBMSSOCMismatch:
		getStringForStateCode := 'BMSSOCMismatch';

	cACBMSVoltageMismatch:
		getStringForStateCode := 'BMSVoltMismatch';

	cACBMSCurrentMismatch:
		getStringForStateCode := 'BMSCurrMismatch';

	cACSensorRangeError:
		getStringForStateCode := 'SensorRange';

	cACHydraulicFilter:
		getStringForStateCode := 'HydFilter';

	cACHydraulicTemperature:
		getStringForStateCode := 'HydTemp';
	
	cACBrakeLowHydraulicPressure:
		getStringForStateCode := 'BrakeHydPress';

	cACOutputFailure:
		getStringForStateCode := 'OutputFailure';
	
	cACDeviceTemperature:
		getStringForStateCode := 'DeviceTemp';

	cACDeviceVoltage:
		getStringForStateCode := 'DeviceVoltage';
		
	cACSoftwareCrash:
		getStringForStateCode := 'SoftwareCrash';

	cACFailSafeMode:
		getStringForStateCode := 'FailSafeMode';
	
	cACMaintenanceMode:
		getStringForStateCode := 'MaintenanceMode';

	cACWatchdogDisabled:
		getStringForStateCode := 'WatchdogDsbld';
		
	cACExecutionFailed:
		getStringForStateCode := 'ExecutionFail';

	cACPersistedCommands:
		getStringForStateCode := 'PersistCmds';
	
	cACSoftware:
		getStringForStateCode := 'Software';

	cACConfiguration:
		getStringForStateCode := 'Configuration';

	cACVoltage:
		getStringForStateCode := 'Voltage';

	cACTemperature:
		getStringForStateCode := 'Temperature';

	cACRelayFuse:
		getStringForStateCode := 'RelayOrFuse';

	cACFuse:
		getStringForStateCode := 'Fuse';

	cACSubsystem:
		getStringForStateCode := 'Subsystem';

	cACConsumable:
		getStringForStateCode := 'Consumable';

	cACHeartbeat:
		getStringForStateCode := 'Heartbeat';

	cACOutput:
		getStringForStateCode := 'Output';

	cACControlSignal:
		getStringForStateCode := 'ControlSignal';
	
	cDCChargerStandby:
		getStringForStateCode := 'ChrgStdby';

	cDCChargerConnected:
		getStringForStateCode := 'ChrgConn';

	cDCChargerDisconnected:
		getStringForStateCode := 'ChrgDiscon';

	cDCTMSCooling:
		getStringForStateCode := 'TMSCooling';

	cDCTMSHeating:
		getStringForStateCode := 'TMSHeating';

	cDCBMSTMSCooling:
		getStringForStateCode := 'BMSTMSCooling';

	cDCBMSTMSHeating:
		getStringForStateCode := 'BMSTMSHeating';

	cDCBMSTMSNoCirculation:
		getStringForStateCode := 'BMSTMSNoCirc';

	cCCChargerStandby:
		getStringForStateCode := 'ChrgStdby';

	cCCChargerConnected:
		getStringForStateCode := 'ChrgConn';

	cCCChargerDisconnected:
		getStringForStateCode := 'ChrgDiscon';

	cCCWaitingForBrakeDisengaged:
		getStringForStateCode := 'WaitBrkDiseng';

	cCCWaitingForParked:
		getStringForStateCode := 'WaitParked';

	cCCCommandStart:
		getStringForStateCode := 'CmdStart';

	cCCCommandStop:
		getStringForStateCode := 'CmdStop';

	cCCStopOnTimeout:
		getStringForStateCode := 'StopOnTimeout';

	cCCLockoutInterlock:
		getStringForStateCode := 'iLockout';

	cCCPosOnlyInterlock:
		getStringForStateCode := 'iPosOnly';

	cCCScaledInterlock:
		getStringForStateCode := 'iScaled';

	cCCThresholdInterlock:
		getStringForStateCode := 'iThreshold';

	cCCSynchronousInterlock:
		getStringForStateCode := 'iSync';

	cCCTwistlocksReadyInterlock:
		getStringForStateCode := 'iTwistRdy';
		
	cCCAutomaticStart:
		getStringForStateCode := 'AutoStart';
		
	cCCSyncState:
		getStringForStateCode := 'SyncState';
		
	cCCCurrentUserNotEnabled:
		getStringForStateCode := 'UserDisabled';
		
	cCCStandby:
		getStringForStateCode := 'Standby';
		
	cCCCycleOutput:
		getStringForStateCode := 'CycleOutput';
END_CASE

IF (strcmp(getStringForStateCode,'state')) THEN
	gStateCodeLastUnknown := code;
END_IF
          
END_FUNCTION

FUNCTION_BLOCK GlobalTypeHandler
  VAR CONSTANT
    cEnumRegisterMax : USINT := ANY_TO_USINT(cEnumTypeDataType);
  END_VAR
  VAR
    lEnumRegister : ARRAY[1..cEnumRegisterMax] OF TypeHandlerEnum;
  END_VAR

            
          

METHOD initialize
  VAR
    ptr : POINTER TO TypeHandlerEnum;
  END_VAR
                  
ptr := ADR(lEnumRegister[cEnumTypeActiveState]);
ptr^.Definition.option := cEnumTypeActiveState;
ptr^.Definition.token := 'active_state';
ptr^.Definition.description := 'States in the Active state machine';
	
ptr^.defineOption(cActiveStateNone,'none','');
ptr^.defineOption(cActiveStatePre,'pre','');
ptr^.defineOption(cActiveStatePost,'post','');
ptr^.defineOption(cActiveStateActive,'active','');

ptr := ADR(lEnumRegister[cEnumTypeBMSChargeState]);
ptr^.Definition.option := cEnumTypeBMSChargeState;
ptr^.Definition.token := 'bms_charge_state';
ptr^.Definition.description := 'States in the BMS charge state machine';
	
ptr^.defineOption(cBMSChargeStateShutdown,'shutdown','');
ptr^.defineOption(cBMSChargeStateDC,'dc','');
ptr^.defineOption(cBMSChargeStateAC,'ac','');
ptr^.defineOption(cBMSChargeStateOther,'other','');

ptr := ADR(lEnumRegister[cEnumTypeBMSFaultLevel]);
ptr^.Definition.option := cEnumTypeBMSFaultLevel;
ptr^.Definition.token := 'bms_fault_level';
ptr^.Definition.description := 'BMS fault level';
	
ptr^.defineOption(cBMSFaultLevelNone,'none','');
ptr^.defineOption(cBMSFaultLevelLow,'low','');
ptr^.defineOption(cBMSFaultLevelMedium,'medium','');
ptr^.defineOption(cBMSFaultLevelSevere,'severe','');

ptr := ADR(lEnumRegister[cEnumTypeBMSState]);
ptr^.Definition.option := cEnumTypeBMSState;
ptr^.Definition.token := 'bms_state';
ptr^.Definition.description := 'States in the BMS state machine';
	
ptr^.defineOption(cBMSStateShutdown,'shutdown','');
ptr^.defineOption(cBMSStateStandby,'standby','');
ptr^.defineOption(cBMSStateDisconnected,'disconnected','');
ptr^.defineOption(cBMSStateConnected,'connected','');

ptr := ADR(lEnumRegister[cEnumTypeChannelMask]);
ptr^.Definition.option := cEnumTypeChannelMask;
ptr^.Definition.token := 'channel_id';
ptr^.Definition.description := 'Channel identifiers (mask)';
	
ptr^.defineOption(cChannelNone,'none','');
ptr^.defineOption(cChannelUIRadio,'Radio','');
ptr^.defineOption(cChannelUICabin,'Cabin','');
ptr^.defineOption(cChannelLogTCP,'Log','');
ptr^.defineOption(cChannelUIRCache,'UIRCache','');
ptr^.defineOption(cChannelMaster,'Master','');
ptr^.defineOption(cChannelEdgeLog,'EdgeLog','');
ptr^.defineOption(cChannelEdgeStateMetric,'EdgeStateMetric','');
ptr^.defineOption(cChannelEdgeValueMetric,'EdgeValueMetric','');
ptr^.defineOption(cChannelEdgeTrace,'EdgeTrace','');

ptr := ADR(lEnumRegister[cEnumTypeChargeQualifier]);
ptr^.Definition.option := cEnumTypeChargeQualifier;
ptr^.Definition.token := 'charge_qualifier';
ptr^.Definition.description := 'Charge modulation qualifier options';
	
ptr^.defineOption(cChargeQualifierBoth,'both','');
ptr^.defineOption(cChargeQualifierCharge,'charge','');
ptr^.defineOption(cChargeQualifierDischarge,'discharge','');
ptr^.defineOption(cChargeQualifierNone,'none','');

ptr := ADR(lEnumRegister[cEnumTypeDataType]);
ptr^.Definition.option := cEnumTypeDataType;
ptr^.Definition.token := 'data_type';
ptr^.Definition.description := 'Native data types';
	
ptr^.defineOption(cDataTypeNone,'none','');
ptr^.defineOption(cDataTypeEnum,'enum','');
ptr^.defineOption(cDataTypeString,'string','');
ptr^.defineOption(cDataTypeUSINT,'usint','');
ptr^.defineOption(cDataTypeUINT,'uint','');
ptr^.defineOption(cDataTypeULINT,'ulint','');
ptr^.defineOption(cDataTypeUDINT,'udint','');
ptr^.defineOption(cDataTypeINT,'int','');
ptr^.defineOption(cDataTypePercentage,'percentage','');
ptr^.defineOption(cDataTypeReal,'real','');
ptr^.defineOption(cDataTypeDWORD,'dword','');
ptr^.defineOption(cDataTypeBool,'bool','');

ptr := ADR(lEnumRegister[cEnumTypeDebugMask]);
ptr^.Definition.option := cEnumTypeDebugMask;
ptr^.Definition.token := 'debug_flag';
ptr^.Definition.description := 'Debug flag (mask)';
	
ptr^.defineOption(cDebugNone,'none','');
ptr^.defineOption(cDebugWaitForLog,'wait_for_log','');
ptr^.defineOption(cDebugEnableFailSafeOnCrash,'enbl_fail_safe','');
ptr^.defineOption(cDebugDisableWatchdog,'dsbl_watch_dog','');
ptr^.defineOption(cDebugSimulateCrash,'simulate_crash','');
ptr^.defineOption(cDebugSimulateA,'simulate_a','');
ptr^.defineOption(cDebugSimulateB,'simulate_b','');
ptr^.defineOption(cDebugSimulateC,'simulate_c','');

ptr := ADR(lEnumRegister[cEnumTypeExecuteOption]);
ptr^.Definition.option := cEnumTypeExecuteOption;
ptr^.Definition.token := 'execute_option';
ptr^.Definition.description := 'Options passed to execution calls';

ptr^.defineOption(cExecuteOptionNone,'none','');
ptr^.defineOption(cExecuteOptionRecurse,'recurse','');
ptr^.defineOption(cExecuteOptionVerbose,'verbose','');
ptr^.defineOption(cExecuteOptionParameter,'parameter','');
ptr^.defineOption(cExecuteOptionSyntax,'syntax','');
ptr^.defineOption(cExecuteOptionChildren,'children','');
ptr^.defineOption(cExecuteOptionExecutor,'executor','');
ptr^.defineOption(cExecuteOptionSubsystems,'subsystems','');
ptr^.defineOption(cExecuteOptionPersist,'persist','');
ptr^.defineOption(cExecuteOptionAll,'all','');
ptr^.defineOption(cExecuteOptionMetadata,'metadata','');

ptr := ADR(lEnumRegister[cEnumTypeExecuteReturn]);
ptr^.Definition.option := cEnumTypeExecuteReturn;
ptr^.Definition.token := 'execute_return';
ptr^.Definition.description := 'Execution exit codes';

ptr^.defineOption(cExecuteReturnOK,'OK','');
ptr^.defineOption(cExecuteReturnUnknownArgumentValue,'bad_arg_value','');
ptr^.defineOption(cExecuteReturnUnsupportedForParticleType,'bad_for_context','');
ptr^.defineOption(cExecuteReturnNullParticle,'null_object','');
ptr^.defineOption(cExecuteReturnSetOverflow,'set_overflow','');
ptr^.defineOption(cExecuteReturnUnknownOption,'bad_option','');	
ptr^.defineOption(cExecuteReturnOKNOK,'returned_NOK','');
ptr^.defineOption(cExecuteReturnUnknownCommand,'bad_command','');
ptr^.defineOption(cExecuteReturnUnknownParameter,'bad_parameter','');
ptr^.defineOption(cExecuteReturnUnsupportedRecurse,'illegal_recurse','');
ptr^.defineOption(cExecuteReturnExecutionQueueOverflow,'queue_overflow','');
ptr^.defineOption(cExecuteReturnExecutionQueueNullParticle,'null_queue_obj','');
ptr^.defineOption(cExecuteReturnParseParameterError,'parameter_syntax','');
ptr^.defineOption(cExecuteReturnUnknownOptionChannelMask,'bad_channel','');
ptr^.defineOption(cExecuteReturnUnknownOptionDebugMask,'bad_debug_flag','');
ptr^.defineOption(cExecuteReturnIllegalIndex,'illegal_index','');
ptr^.defineOption(cExecuteReturnMissingArgument,'missing_arg','');
ptr^.defineOption(cExecuteReturnTooFewArguments,'missing_args','');
ptr^.defineOption(cExecuteReturnTooManyArguments,'extra_args','');
ptr^.defineOption(cExecuteReturnInternalError,'internal','');
ptr^.defineOption(cExecuteReturnPersistFailed,'persist_failed','');
ptr^.defineOption(cExecuteReturnUnprocessedArguments,'unproc_args','');
ptr^.defineOption(cExecuteReturnExecutionExecutorFailed,'monitor_failed','');
ptr^.defineOption(cExecuteReturnExecutionSyntax,'syntax_error','');
ptr^.defineOption(cExecuteReturnExecutionSyntaxIncompleteRequest,'incmplt_reqst','');
ptr^.defineOption(cExecuteReturnExecutionSyntaxIncompleteParameter,'incmplt_prm','');
ptr^.defineOption(cExecuteReturnExecutionSyntaxIncompleteName,'incmplt_name','');
ptr^.defineOption(cExecuteReturnExecutionSyntaxTokenOverflow,'token_overflow','');
ptr^.defineOption(cExecuteReturnExecutionSyntaxStartWithName,'start_name','');
ptr^.defineOption(cExecuteReturnExecutionSyntaxCommandAfterName,'name_then_cmd','');
ptr^.defineOption(cExecuteReturnExecutionSyntaxDuplicateCommands,'duplicate_cmd','');
ptr^.defineOption(cExecuteReturnExecutionSyntaxUnkownName,'unknown_name','');
ptr^.defineOption(cExecuteReturnExecutionSyntaxUnkownNameForParameter,'unkn_name_par','');
ptr^.defineOption(cExecuteReturnExecutionSyntaxTooManyOptions,'excess_options','');
ptr^.defineOption(cExecuteReturnExecutionSyntaxUnbounded,'syntax_unbounded','');
ptr^.defineOption(cExecuteReturnReadOnly,'read_only','');

ptr := ADR(lEnumRegister[cEnumTypeFunctionalMode]);
ptr^.Definition.option := cEnumTypeFunctionalMode;
ptr^.Definition.token := 'functional_mode';
ptr^.Definition.description := 'Machine functional mode';

ptr^.defineOption(cFunctionalModeAny,'any','');
ptr^.defineOption(cFunctionalModeDefault,'default','');
ptr^.defineOption(cFunctionalModeTravel,'travel','');
ptr^.defineOption(cFunctionalModeLift,'lift','');
ptr^.defineOption(cFunctionalModeSpreaderConfiguration,'sprd_cnfg','');
ptr^.defineOption(cFunctionalModeTopbeamConfiguration,'topbm_cnfg','');

ptr := ADR(lEnumRegister[cEnumTypeInputMode]);
ptr^.Definition.option := cEnumTypeInputMode;
ptr^.Definition.token := 'input_mode';
ptr^.Definition.description := 'Machine input mode';
	
ptr^.defineOption(cInputModeNone,'none','');
ptr^.defineOption(cInputModeDefault,'default','');
ptr^.defineOption(cInputModeSpreaderConfiguration,'sprd_cnfg','');
ptr^.defineOption(cInputModeTopbeamConfiguration,'topbm_cnfg','');

ptr := ADR(lEnumRegister[cEnumTypeLockState]);
ptr^.Definition.option := cEnumTypeLockState;
ptr^.Definition.token := 'lock_state';
ptr^.Definition.description := 'Twistlock lock state';

ptr^.defineOption(cLockStateNone,'none','');
ptr^.defineOption(cLockStateUnlocked,'unlocked','');
ptr^.defineOption(cLockStateLocked,'locked','');
ptr^.defineOption(cLockStatePartial,'partial','');

ptr := ADR(lEnumRegister[cEnumTypeOBCState]);
ptr^.Definition.option := cEnumTypeOBCState;
ptr^.Definition.token := 'obc_state';
ptr^.Definition.description := 'Onboard charger state';

ptr^.defineOption(cOBCStateDisconnected,'disconnect','');
ptr^.defineOption(cOBCStateCharging,'charging','');
ptr^.defineOption(cOBCStateStandby,'standby','');
ptr^.defineOption(cOBCStateError,'error','');

ptr := ADR(lEnumRegister[cEnumTypeOBCStatus]);
ptr^.Definition.option := cEnumTypeOBCStatus;
ptr^.Definition.token := 'obc_status';
ptr^.Definition.description := 'Onboard charger status';

ptr^.defineOption(cOBCStatusNone,'none','');
ptr^.defineOption(cOBCStatusCharging,'charging','');
ptr^.defineOption(cOBCStatusStandby,'standby','');
ptr^.defineOption(cOBCStatusError,'error','');

ptr := ADR(lEnumRegister[cEnumTypeOperatingMethod]);
ptr^.Definition.option := cEnumTypeOperatingMethod;
ptr^.Definition.token := 'operating_method';
ptr^.Definition.description := 'Operating mode commands';

ptr^.defineOption(cOperatingMethodNone,'none','');
ptr^.defineOption(cOperatingMethodPark,'park','');
ptr^.defineOption(cOperatingMethodUnpark,'unpark','');
ptr^.defineOption(cOperatingMethodLock,'lock','');
ptr^.defineOption(cOperatingMethodLockWithoutPark,'lock_no_park','');
ptr^.defineOption(cOperatingMethodUnlock,'unlock','');
ptr^.defineOption(cOperatingMethodSlow,'slow','');
ptr^.defineOption(cOperatingMethodNormal,'normal','');

ptr := ADR(lEnumRegister[cEnumTypeProgMovCode]);
ptr^.Definition.option := cEnumTypeProgMovCode;
ptr^.Definition.token := 'progmov_code';
ptr^.Definition.description := 'Automation code';

ptr^.defineOption(cProgMovCodeNone,'none','');
ptr^.defineOption(cProgMovCode_Steer_0,'steer_0','');

ptr := ADR(lEnumRegister[cEnumTypeRunState]);
ptr^.Definition.option := cEnumTypeRunState;
ptr^.Definition.token := 'run_state';
ptr^.Definition.description := 'Run state machine';

ptr^.defineOption(cRunStateNone,'none','');
ptr^.defineOption(cRunStateStart,'start','');
ptr^.defineOption(cRunStateStop,'stop','');

ptr := ADR(lEnumRegister[cEnumTypeSeverity]);
ptr^.Definition.option := cEnumTypeSeverity;
ptr^.Definition.token := 'severity';
ptr^.Definition.description := 'Severity options';

ptr^.defineOption(cSeverityNone,'none','');
ptr^.defineOption(cSeverityWarning,'warning','');
ptr^.defineOption(cSeverityError,'error','');
ptr^.defineOption(cSeverityCritical,'critical','');

ptr := ADR(lEnumRegister[cEnumTypeShutdownCode]);
ptr^.Definition.option := cEnumTypeShutdownCode;
ptr^.Definition.token := 'shutdown_code';
ptr^.Definition.description := 'Device shutdown diagnostic';

ptr^.defineOption(cShutdownCodeUnknown,'unknown','');
ptr^.defineOption(cShutdownCodeIgnition,'ignition','');
ptr^.defineOption(cShutdownCodeSoftware,'software','');
ptr^.defineOption(cShutdownCodeSupervisor,'supervisor','');
ptr^.defineOption(cShutdownCodeCrashDetected,'crash','');
ptr^.defineOption(cShutdownCodeTrapDetected,'trap','');

ptr := ADR(lEnumRegister[cEnumTypeSteerMode]);
ptr^.Definition.option := cEnumTypeSteerMode;
ptr^.Definition.token := 'steer_mode';
ptr^.Definition.description := 'Steering modes';

ptr^.defineOption(cSteerModeNone,'none','');
ptr^.defineOption(cSteerMode4WS,'4ws','');
ptr^.defineOption(cSteerModeLateral,'lateral','');
ptr^.defineOption(cSteerModeCarousel,'carousel','');
ptr^.defineOption(cSteerModeReconfigure,'reconfigure','');
ptr^.defineOption(cSteerModeLateralNeg90,'lat_neg_90','');
ptr^.defineOption(cSteerModeLateralPos90,'lat_pos_90','');
ptr^.defineOption(cSteerModeCustom,'custom','');

ptr := ADR(lEnumRegister[cEnumTypeSubsystem]);
ptr^.Definition.option := cEnumTypeSubsystem;
ptr^.Definition.token := 'subsystem';
ptr^.Definition.description := 'Machine subsystems';

ptr^.defineOption(cSubsystemNone,'none','');
ptr^.defineOption(cSubsystemSpreader,'Spreader','');
ptr^.defineOption(cSubsystemBeacons,'Beacons','');
ptr^.defineOption(cSubsystemCabin,'Cabin','');
ptr^.defineOption(cSubsystemLights,'Lights','');
ptr^.defineOption(cSubsystemPowerpack,'owerpack','');
ptr^.defineOption(cSubsystemSideshiftAB,'SideshiftAB','');
ptr^.defineOption(cSubsystemSideshiftCD,'SideshiftCD','');
ptr^.defineOption(cSubsystemSpreaderPowerPack,'SprPowerPack','');
ptr^.defineOption(cSubsystemSteerA,'SteerA','');
ptr^.defineOption(cSubsystemSteerB,'SteerB','');
ptr^.defineOption(cSubsystemSteerC,'SteerC','');
ptr^.defineOption(cSubsystemSteerD,'SteerD','');
ptr^.defineOption(cSubsystemTravelA,'TravelA','');
ptr^.defineOption(cSubsystemTravelB,'TravelB','');
ptr^.defineOption(cSubsystemTravelC,'TravelC','');
ptr^.defineOption(cSubsystemTravelD,'TravelD','');
ptr^.defineOption(cSubsystemWinchA,'WinchA','');
ptr^.defineOption(cSubsystemWinchB,'WinchB','');
ptr^.defineOption(cSubsystemWinchC,'WinchC','');
ptr^.defineOption(cSubsystemWinchD,'WinchD','');
ptr^.defineOption(cSubsystemTwistlockA,'TwistlockA','');
ptr^.defineOption(cSubsystemTwistlockB,'TwistlockB','');
ptr^.defineOption(cSubsystemTwistlockC,'TwistlockC','');
ptr^.defineOption(cSubsystemTwistlockD,'TwistlockD','');
ptr^.defineOption(cSubsystemTopbeamAB,'TopbeamAB','');
ptr^.defineOption(cSubsystemTopbeamCD,'TopbeamCD','');
ptr^.defineOption(cSubsystemCANBusSystem,'CANBusSystem','');
ptr^.defineOption(cSubsystemCANBusDrive,'CANBusDrive','');
ptr^.defineOption(cSubsystemBattery,'Battery','');
ptr^.defineOption(cSubsystemSecondary,'Secondary','');
ptr^.defineOption(cSubsystemUInterface,'UInterface','');
ptr^.defineOption(cSubsystemHydraulics,'Hydraulics','');
ptr^.defineOption(cSubsystemLift,'Lift','');
ptr^.defineOption(cSubsystemTravel,'Travel','');
ptr^.defineOption(cSubsystemSteer,'Steer','');
ptr^.defineOption(cSubsystemMachine,'Machine','');

ptr := ADR(lEnumRegister[cEnumTypeSystemControl]);
ptr^.Definition.option := cEnumTypeSystemControl;
ptr^.Definition.token := 'system_control';
ptr^.Definition.description := 'Options for controlling system state';

ptr^.defineOption(cSystemControlReset,'reset','');
ptr^.defineOption(cSystemControlEStop,'estop','');
ptr^.defineOption(cSystemControlStop,'stop','');
ptr^.defineOption(cSystemControlStart,'start','');
ptr^.defineOption(cSystemControlNone,'none','');

ptr := ADR(lEnumRegister[cEnumTypeSystemState]);
ptr^.Definition.option := cEnumTypeSystemState;
ptr^.Definition.token := 'system_state';
ptr^.Definition.description := 'System state machine';

ptr^.defineOption(cSystemStateNone,'none','');
ptr^.defineOption(cSystemStateInitialized,'initialized','');
ptr^.defineOption(cSystemStateStandby,'standby','');
ptr^.defineOption(cSystemStatePreparing,'preparing','');
ptr^.defineOption(cSystemStateCharging,'charging','');
ptr^.defineOption(cSystemStatePreOperational,'pre_operational','');
ptr^.defineOption(cSystemStatePoweringDown,'powering_down','');
ptr^.defineOption(cSystemStatePoweringUp,'powering_up','');
ptr^.defineOption(cSystemStateGoOperational,'go_operational','');
ptr^.defineOption(cSystemStateExitOperational,'exit_operational','');
ptr^.defineOption(cSystemStateOperational,'operational','');

ptr := ADR(lEnumRegister[cEnumTypeTMSState]);
ptr^.Definition.option := cEnumTypeTMSState;
ptr^.Definition.token := 'tms_state';
ptr^.Definition.description := 'Battery thermal management state';

ptr^.defineOption(cTMSStateShutdown,'shutdown','');
ptr^.defineOption(cTMSStateCooling,'cooling','');
ptr^.defineOption(cTMSStateHeating,'heating','');
ptr^.defineOption(cTMSStateCirculation,'circulation','');

ptr := ADR(lEnumRegister[cEnumTypeTokenType]);
ptr^.Definition.option := cEnumTypeTokenType;
ptr^.Definition.token := 'token_type';
ptr^.Definition.description := 'Standard tokens';

ptr^.defineOption(cTokenNone,'none','');
ptr^.defineOption(cTokenDescribe,'describe','');
ptr^.defineOption(cTokenSyntax,'syntax','');
ptr^.defineOption(cTokenVerify,'verify','');
ptr^.defineOption(cTokenIdentify,'identify','');
ptr^.defineOption(cTokenRegister,'register','');
ptr^.defineOption(cTokenConfigure,'configure','');
ptr^.defineOption(cTokenSetFailSafeMode,'failsafe_set','');
ptr^.defineOption(cTokenClearFailSafeMode,'failsafe_clr','');
ptr^.defineOption(cTokenFailSafeConfig,'failsafe_cnfg','');
ptr^.defineOption(cTokenProceed,'proceed','');
ptr^.defineOption(cTokenList,'list','');
ptr^.defineOption(cTokenDebugMaskAdd,'debug_add','');
ptr^.defineOption(cTokenDebugMaskDelete,'debug_del','');
ptr^.defineOption(cTokenDebugMaskClear,'debug_clr','');
ptr^.defineOption(cTokenClose,'close','');
ptr^.defineOption(cTokenExport,'export','');
ptr^.defineOption(cTokenClear,'clear','');
ptr^.defineOption(cTokenDeregister,'deregister','');
ptr^.defineOption(cTokenTrigger,'trigger','');
ptr^.defineOption(cTokenChannelMaskAdd,'chanmask_add','');
ptr^.defineOption(cTokenChannelMaskDelete,'chanmask_del','');
ptr^.defineOption(cTokenChannelMaskClear,'chanmask_clr','');
ptr^.defineOption(cTokenChannelIndex,'channel','');
ptr^.defineOption(cTokenValue,'value','');
ptr^.defineOption(cTokenOverrideValue,'override_value','');
ptr^.defineOption(cTokenOverride,'override','');
ptr^.defineOption(cTokenValueType,'value_type','');
ptr^.defineOption(cTokenMeaning,'meaning','');
ptr^.defineOption(cTokenOverrideMeaning,'override_meaning','');
ptr^.defineOption(cTokenRawIndex,'raw_index','');
ptr^.defineOption(cTokenIndex,'index','');
ptr^.defineOption(cTokenUnknown,'unknown','');
ptr^.defineOption(cTokenObject,'object','');
ptr^.defineOption(cTokenFeature,'arg','');
ptr^.defineOption(cTokenZero,'zero','');
ptr^.defineOption(sTokenUpper,'upper','');
ptr^.defineOption(cTokenThreshold,'threshold','');
ptr^.defineOption(cTokenHysteresis,'hysteresis','');
ptr^.defineOption(cTokenImport,'import','');

ptr := ADR(lEnumRegister[cEnumTypeUiEventCode]);
ptr^.Definition.option := cEnumTypeUiEventCode;
ptr^.Definition.token := 'ui_event_code';
ptr^.Definition.description := 'User Interface event code';

ptr^.defineOption(cUIEventCodeNone,'none','');
ptr^.defineOption(cUIEventCodeToggleLights,'toggle_lights','');
ptr^.defineOption(cUIEventCodeUIModeResponse,'ui_mode_resp','');
ptr^.defineOption(cUIEventCodeToggleSpreaderConfiguration,'sprd_cnfg','');
ptr^.defineOption(cUIEventCodeSpreaderExtensionAutoCommand,'sprd_extend','');
ptr^.defineOption(cUIEventCodeSpreaderRetractionAutoCommand,'sprd_retract','');
ptr^.defineOption(cUIEventCodeInitiate,'initiate','');
ptr^.defineOption(cUIEventCodeStart,'start','');
ptr^.defineOption(cUIEventCodeStop,'stop','');
ptr^.defineOption(cUIEventCodeProgMovStart,'prog_move_start','');

ptr := ADR(lEnumRegister[cEnumTypeUiOrientation]);
ptr^.Definition.option := cEnumTypeUiOrientation;
ptr^.Definition.token := 'ui_orientation';
ptr^.Definition.description := 'User Interface orientation';

ptr^.defineOption(cUIOrientationNone,'none','');
ptr^.defineOption(cUIOrientationForward,'forward','');
ptr^.defineOption(cUIOrientationSide,'side','');
ptr^.defineOption(cUIOrientationReverse,'reverse','');
ptr^.defineOption(cUIOrientationOpposite,'opposite','');

ptr := ADR(lEnumRegister[cEnumTypeValueStyle]);
ptr^.Definition.option := cEnumTypeValueStyle;
ptr^.Definition.token := 'value_style';
ptr^.Definition.description := 'How a value is treated';

ptr^.defineOption(cValueStyleConfigurable,'configurable','');
ptr^.defineOption(cValueStyleParameter,'parameter','');
ptr^.defineOption(cValueStyleTrigger,'trigger','');

(*registerEnum(ADR(sEnumBMSChargeState));
registerEnum(ADR(sEnumBMSFaultLevel));
registerEnum(ADR(sEnumBMSState));
registerEnum(ADR(sEnumChannelMask));
registerEnum(ADR(sEnumChargeQualifier));
registerEnum(ADR(sEnumDebugMask));
registerEnum(ADR(sEnumDataType));
registerEnum(ADR(sEnumExecuteOption));
registerEnum(ADR(sEnumExecuteReturn));
registerEnum(ADR(sEnumFunctionalMode));
registerEnum(ADR(sEnumInputMode));
registerEnum(ADR(sEnumLockState));
registerEnum(ADR(sEnumOBCState));
registerEnum(ADR(sEnumOBCStatus));
registerEnum(ADR(sEnumOperatingMethod));
registerEnum(ADR(sEnumRunState));
registerEnum(ADR(sEnumSeverity));
registerEnum(ADR(sEnumShutdownCode));
registerEnum(ADR(sEnumSteerMode));
registerEnum(ADR(sEnumSubsystem));
registerEnum(ADR(sEnumSystemControl));
registerEnum(ADR(sEnumSystemState));
registerEnum(ADR(sEnumTMSState));
registerEnum(ADR(sEnumTokenType));
registerEnum(ADR(sEnumUIEventCode));
registerEnum(ADR(sEnumUIOrientation));
registerEnum(ADR(sEnumValueStyle));*)

// simulation code space
// base 456332
// defineOption_1(0,'','');
// option description t_long_string to t_short_string: no change
// reduce ptr^.defineOption(): 100 bytes per call
// reduce customer type handler: 1500bytes per handler based on bmschargestate

// gSystem: move to pointers = 455700, not much change as not much duplication

// v5: 453712 gSystem is not pointers but in code space
// 454584: derive EC classes for monitor and parse, 400bytes each
// 454518: ready for testing
                
END_METHOD

METHOD getBoolFromToken : BOOL
  VAR_INPUT
    token : t_token_string;
    target : REFERENCE TO BOOL;
  END_VAR
                  getBoolFromToken := sTypeHandlerBool.getValue(token,target);

                
END_METHOD

METHOD getDWORDFromToken : BOOL
  VAR_INPUT
    token : t_token_string;
    target : REFERENCE TO DWORD;
  END_VAR
                  getDWORDFromToken := sTypeHandlerDWORD.getValue(token,target);

                
END_METHOD

METHOD registerEnum
  VAR_INPUT
    handler : POINTER TO TypeHandlerEnum;
  END_VAR
  VAR
    index : INT;
  END_VAR
                  IF (handler=0) THEN
	RETURN;
END_IF

index := handler^.Definition.option;

IF ((index>cEnumRegisterMax) OR
	(index<0)) THEN
	gCodeErrorHandler(pMessage:='EnumRegister definition out of bounds');
	RETURN;
END_IF

IF ((lEnumRegister[index]<>0) AND
	(lEnumRegister[index]<>handler)) THEN
	gCodeErrorHandler(pMessage:='EnumRegister already registered');
	RETURN;
END_IF

IF (lEnumRegister[index]=0) THEN
	lEnumRegister[index] := handler;
END_IF

handler^.initialize();

                
END_METHOD

METHOD getTokenForEnum : t_token_string
  VAR_INPUT
    enumType : INT;
    value : INT;
  END_VAR
                  IF ((enumType<=0) OR
	(enumType>cEnumRegisterMax)) THEN
	getTokenForEnum := 'illegal';
	RETURN;
END_IF

getTokenForEnum := lEnumRegister[enumType].getToken(value);

                
END_METHOD

METHOD getEnumFromToken : BOOL
  VAR_INPUT
    enumType : INT;
    token : t_token_string;
    target : REFERENCE TO INT;
  END_VAR
  VAR
    i : USINT;
  END_VAR
                  IF ((enumType>cEnumRegisterMax) OR
	(enumType<=0)) THEN

	getEnumFromToken := FALSE;
	
	RETURN;
END_IF

getEnumFromToken := lEnumRegister[enumType].getValue(token,target);

                
END_METHOD

METHOD getTokenForPercentage : t_token_string
  VAR_INPUT
    value : t_percentage;
  END_VAR
                  getTokenForPercentage := sTypeHandlerPercentage.getToken(value);
                
END_METHOD

METHOD getTokenForREAL : t_token_string
  VAR_INPUT
    value : REAL;
  END_VAR
                  getTokenForREAL := sTypeHandlerREAL.getToken(value);
                
END_METHOD

METHOD getTokenForDWORD : t_token_string
  VAR_INPUT
    value : DWORD;
  END_VAR
                  getTokenForDWORD := sTypeHandlerDWORD.getToken(value);
                
END_METHOD

METHOD getTokenForBool : t_token_string
  VAR_INPUT
    value : BOOL;
  END_VAR
                  getTokenForBool := sTypeHandlerBool.getToken(value);
                
END_METHOD

METHOD getTokenForINT : t_token_string
  VAR_INPUT
    value : INT;
  END_VAR
                  getTokenForINT := sTypeHandlerINT.getToken(value);
                
END_METHOD

METHOD getTokenForUDINT : t_token_string
  VAR_INPUT
    value : UDINT;
  END_VAR
                  getTokenForUDINT := sTypeHandlerUDINT.getToken(value);
                
END_METHOD

METHOD getTokenForULINT : t_token_string
  VAR_INPUT
    value : ULINT;
  END_VAR
                  getTokenForULINT := sTypeHandlerULINT.getToken(value);
                
END_METHOD

METHOD getTokenForUSINT : t_token_string
  VAR_INPUT
    value : USINT;
  END_VAR
                  getTokenForUSINT := sTypeHandlerUSINT.getToken(value);
                
END_METHOD

METHOD getTokenForUINT : t_token_string
  VAR_INPUT
    value : UINT;
  END_VAR
                  getTokenForUINT := sTypeHandlerUINT.getToken(value);
                
END_METHOD

METHOD getTokenForEnumType : t_token_string
  VAR_INPUT
    enumType : t_enum_type;
  END_VAR
                  IF ((enumType<=0) OR
	(enumType>cEnumRegisterMax)) THEN
	getTokenForEnumType := 'illegal';
	RETURN;
END_IF

getTokenForEnumType := lEnumRegister[enumType].Definition.token;

                
END_METHOD

METHOD getTokenForDataType : t_token_string
  VAR_INPUT
    dataType : t_data_type;
  END_VAR
                  getTokenForDataType := getTokenForEnum(cEnumTypeDataType,dataType);

                
END_METHOD

METHOD getREALFromToken : BOOL
  VAR_INPUT
    token : t_token_string;
    target : REFERENCE TO REAL;
  END_VAR
                  getREALFromToken := sTypeHandlerREAL.getValue(token,target);

                
END_METHOD

METHOD getPercentageFromToken : BOOL
  VAR_INPUT
    token : t_token_string;
    target : REFERENCE TO t_percentage;
  END_VAR
                  getPercentageFromToken := sTypeHandlerPercentage.getValue(token,target);

                
END_METHOD

METHOD getINTFromToken : BOOL
  VAR_INPUT
    token : t_token_string;
    target : REFERENCE TO INT;
  END_VAR
                  getINTFromToken := sTypeHandlerINT.getValue(token,target);

                
END_METHOD

METHOD getUSINTFromToken : BOOL
  VAR_INPUT
    token : t_token_string;
    target : REFERENCE TO USINT;
  END_VAR
                  getUSINTFromToken := sTypeHandlerUSINT.getValue(token,target);

                
END_METHOD

METHOD getUINTFromToken : BOOL
  VAR_INPUT
    token : t_token_string;
    target : REFERENCE TO UINT;
  END_VAR
                  getUINTFromToken := sTypeHandlerUINT.getValue(token,target);

                
END_METHOD

METHOD getULINTFromToken : BOOL
  VAR_INPUT
    token : t_token_string;
    target : REFERENCE TO ULINT;
  END_VAR
                  getULINTFromToken := sTypeHandlerULINT.getValue(token,target);

                
END_METHOD

METHOD getUDINTFromToken : BOOL
  VAR_INPUT
    token : t_token_string;
    target : REFERENCE TO UDINT;
  END_VAR
                  getUDINTFromToken := sTypeHandlerUDINT.getValue(token,target);

                
END_METHOD

METHOD getStringForEnumOptions : STRING
  VAR_INPUT
    enumType : t_enum_type;
  END_VAR
  VAR
    str : STRING;
  END_VAR
                  IF ((enumType<=0) OR
	(enumType>cEnumRegisterMax)) THEN
	getStringForEnumOptions := '[]';
	RETURN;
END_IF

getStringForEnumOptions := lEnumRegister[enumType].getOptions();
                
END_METHOD
END_FUNCTION_BLOCK

FUNCTION_BLOCK TypeHandlerBool
  VAR
    lDataType : t_data_type := cDataTypeBool;
  END_VAR

            
          

METHOD getValue : BOOL
  VAR_INPUT
    token : t_token_string;
    target : REFERENCE TO BOOL;
  END_VAR
                  IF ((strcmp(token,'true')) OR
	(strcmp(token,'TRUE'))) THEN
	target := TRUE;
	getValue := TRUE;
	RETURN;
END_IF

IF ((strcmp(token,'false')) OR
	(strcmp(token,'FALSE'))) THEN
	target := FALSE;
	getValue := TRUE;
	RETURN;
END_IF

getValue := FALSE;

                
END_METHOD

METHOD getToken : t_token_string
  VAR_INPUT
    value : BOOL;
  END_VAR
                  IF (value) THEN
	getToken := 'true';
ELSE
	getToken := 'false';
END_IF


                
END_METHOD
END_FUNCTION_BLOCK

FUNCTION_BLOCK TypeHandlerDWORD
  VAR
    lDataType : t_data_type := cDataTypeDWORD;
  END_VAR

            
          

METHOD getValue : BOOL
  VAR_INPUT
    token : t_token_string;
    target : REFERENCE TO DWORD;
  END_VAR
  VAR
    value : DWORD;
  END_VAR
                  value := STRING_TO_DWORD(token);

getValue := strcmp(DWORD_TO_STRING(value),token);
IF (getValue) THEN
	target := value;
END_IF


                
END_METHOD

METHOD getToken : t_token_string
  VAR_INPUT
    value : DWORD;
  END_VAR
                  getToken := DWORD_TO_STRING(value);

                
END_METHOD
END_FUNCTION_BLOCK

FUNCTION_BLOCK TypeHandlerINT
  VAR
    lDataType : t_data_type := cDataTypeINT;
  END_VAR

            
          

METHOD getValue : BOOL
  VAR_INPUT
    token : t_token_string;
    target : REFERENCE TO INT;
  END_VAR
  VAR
    value : INT;
  END_VAR
                  value := STRING_TO_INT(token);

getValue := strcmp(INT_TO_STRING(value),token);
IF (getValue) THEN
	target := value;
END_IF


                
END_METHOD

METHOD getToken : t_token_string
  VAR_INPUT
    value : INT;
  END_VAR
                  getToken := INT_TO_STRING(value);

                
END_METHOD
END_FUNCTION_BLOCK

FUNCTION_BLOCK TypeHandlerPercentage
  VAR
    lDataType : t_data_type := cDataTypePercentage;
  END_VAR

            
          

METHOD getValue : BOOL
  VAR_INPUT
    token : t_token_string;
    target : REFERENCE TO t_percentage;
  END_VAR
  VAR
    value : t_percentage;
  END_VAR
                  value := STRING_TO_REAL(token);

getValue := strcmp(REAL_TO_STRING(value),token);
IF (getValue) THEN
	target := value;
END_IF



                
END_METHOD

METHOD getToken : t_token_string
  VAR_INPUT
    value : t_percentage;
  END_VAR
                  getToken := CONCAT(INT_TO_STRING(REAL_TO_INT(value*100.0)),'%');

                
END_METHOD
END_FUNCTION_BLOCK

FUNCTION_BLOCK TypeHandlerREAL
  VAR
    lDataType : t_data_type := cDataTypeREAL;
  END_VAR

            
          

METHOD getValue : BOOL
  VAR_INPUT
    token : t_token_string;
    target : REFERENCE TO REAL;
  END_VAR
  VAR
    value : REAL;
  END_VAR
                  value := STRING_TO_REAL(token);

getValue := strcmp(REAL_TO_STRING(value),token);
IF (getValue) THEN
	target := value;
END_IF



                
END_METHOD

METHOD getToken : t_token_string
  VAR_INPUT
    value : REAL;
  END_VAR
                  getToken := REAL_TO_STRING(value);

                
END_METHOD
END_FUNCTION_BLOCK

FUNCTION_BLOCK TypeHandlerUDINT
  VAR
    lDataType : t_data_type := cDataTypeUDINT;
  END_VAR

            
          

METHOD getValue : BOOL
  VAR_INPUT
    token : t_token_string;
    target : REFERENCE TO UDINT;
  END_VAR
  VAR
    value : UDINT;
  END_VAR
                  value := STRING_TO_UDINT(token);

getValue := strcmp(UDINT_TO_STRING(value),token);
IF (getValue) THEN
	target := value;
END_IF



                
END_METHOD

METHOD getToken : t_token_string
  VAR_INPUT
    value : UDINT;
  END_VAR
                  getToken := UDINT_TO_STRING(value);

                
END_METHOD
END_FUNCTION_BLOCK

FUNCTION_BLOCK TypeHandlerUINT
  VAR
    lDataType : t_data_type := cDataTypeUINT;
  END_VAR

            
          

METHOD getValue : BOOL
  VAR_INPUT
    token : t_token_string;
    target : REFERENCE TO UINT;
  END_VAR
  VAR
    value : UINT;
  END_VAR
                  value := STRING_TO_UINT(token);

getValue := strcmp(UINT_TO_STRING(value),token);
IF (getValue) THEN
	target := value;
END_IF



                
END_METHOD

METHOD getToken : t_token_string
  VAR_INPUT
    value : UINT;
  END_VAR
                  getToken := UINT_TO_STRING(value);

                
END_METHOD
END_FUNCTION_BLOCK

FUNCTION_BLOCK TypeHandlerULINT
  VAR
    lDataType : t_data_type := cDataTypeULINT;
  END_VAR

            
          

METHOD getValue : BOOL
  VAR_INPUT
    token : t_token_string;
    target : REFERENCE TO ULINT;
  END_VAR
  VAR
    value : ULINT;
  END_VAR
                  value := STRING_TO_ULINT(token);

getValue := strcmp(ULINT_TO_STRING(value),token);
IF (getValue) THEN
	target := value;
END_IF



                
END_METHOD

METHOD getToken : t_token_string
  VAR_INPUT
    value : ULINT;
  END_VAR
                  getToken := ULINT_TO_STRING(value);

                
END_METHOD
END_FUNCTION_BLOCK

FUNCTION_BLOCK TypeHandlerUSINT
  VAR
    lDataType : t_data_type := cDataTypeUSINT;
  END_VAR

            
          

METHOD getValue : BOOL
  VAR_INPUT
    token : t_token_string;
    target : REFERENCE TO USINT;
  END_VAR
  VAR
    value : USINT;
  END_VAR
                  value := STRING_TO_USINT(token);

getValue := strcmp(USINT_TO_STRING(value),token);
IF (getValue) THEN
	target := value;
END_IF



                
END_METHOD

METHOD getToken : t_token_string
  VAR_INPUT
    value : USINT;
  END_VAR
                  getToken := USINT_TO_STRING(value);

                
END_METHOD
END_FUNCTION_BLOCK

FUNCTION getEnumTypeFromToken : t_enum_type
  VAR_INPUT
    token : t_token_string;
    default : INT;
    parseOK : REFERENCE TO BOOL;
  END_VAR

            IF (strcmp(token,'int')) THEN
	getEnumTypeFromToken := cEnumTypeNone;
	RETURN;
END_IF

IF (strcmp(token, 'active_state')) THEN
	getEnumTypeFromToken := cEnumTypeActiveState;
	RETURN;
END_IF

IF (strcmp(token, 'BMS_charge_state')) THEN
	getEnumTypeFromToken := cEnumTypeBMSChargeState;
	RETURN;
END_IF

IF (strcmp(token, 'BMS_fault_level')) THEN
	getEnumTypeFromToken := cEnumTypeBMSFaultLevel;
	RETURN;
END_IF
		
IF (strcmp(token, 'BMS_state')) THEN
	getEnumTypeFromToken := cEnumTypeBMSState;
	RETURN;
END_IF
		
IF (strcmp(token, 'channel_mask')) THEN
	getEnumTypeFromToken := cEnumTypeChannelMask;
	RETURN;
END_IF
		
IF (strcmp(token, 'charge_qualifier')) THEN
	getEnumTypeFromToken := cEnumTypeChargeQualifier;
	RETURN;
END_IF

IF (strcmp(token, 'debug_mask')) THEN
	getEnumTypeFromToken := cEnumTypeDebugMask;
	RETURN;
END_IF
		
IF (strcmp(token, 'event_code')) THEN
	getEnumTypeFromToken := cEnumTypeEventCode;
	RETURN;
END_IF

IF (strcmp(token, 'functional_mode')) THEN
	getEnumTypeFromToken := cEnumTypeFunctionalMode;
	RETURN;
END_IF
		
IF (strcmp(token, 'input_mode')) THEN
	getEnumTypeFromToken := cEnumTypeInputMode;
	RETURN;
END_IF
		
IF (strcmp(token, 'interlock_state')) THEN
	getEnumTypeFromToken := cEnumTypeInterlockState;
	RETURN;
END_IF

IF (strcmp(token, 'lock_state')) THEN
	getEnumTypeFromToken := cEnumTypeLockState;
	RETURN;
END_IF	

IF (strcmp(token, 'OBC_state')) THEN
	getEnumTypeFromToken := cEnumTypeOBCState;
	RETURN;
END_IF
		
IF (strcmp(token, 'OBC_status')) THEN
	getEnumTypeFromToken := cEnumTypeOBCStatus;
	RETURN;
END_IF
		
IF (strcmp(token, 'operating_method')) THEN
	getEnumTypeFromToken := cEnumTypeOperatingMethod;
	RETURN;
END_IF
		
IF (strcmp(token, 'prog_mov_code')) THEN
	getEnumTypeFromToken := cEnumTypeProgMovCode;
	RETURN;
END_IF
		
IF (strcmp(token, 'run_state')) THEN
	getEnumTypeFromToken := cEnumTypeRunState;
	RETURN;
END_IF
		
IF (strcmp(token, 'severity')) THEN
	getEnumTypeFromToken := cEnumTypeSeverity;
	RETURN;
END_IF

IF (strcmp(token, 'shutdown_code')) THEN
	getEnumTypeFromToken := cEnumTypeShutdownCode;
	RETURN;
END_IF

IF (strcmp(token, 'state_code')) THEN
	getEnumTypeFromToken := cEnumTypeStateCode;
	RETURN;
END_IF

IF (strcmp(token, 'steer_mode')) THEN
	getEnumTypeFromToken := cEnumTypeSteerMode;
	RETURN;
END_IF
		
IF (strcmp(token, 'subsystem')) THEN
	getEnumTypeFromToken := cEnumTypeSubsystem;
	RETURN;
END_IF

IF (strcmp(token, 'system_control')) THEN
	getEnumTypeFromToken := cEnumTypeSystemControl;
	RETURN;
END_IF

IF (strcmp(token, 'system_state')) THEN
	getEnumTypeFromToken := cEnumTypeSystemState;
	RETURN;
END_IF
		
IF (strcmp(token, 'TMS_state')) THEN
	getEnumTypeFromToken := cEnumTypeTMSState;
	RETURN;
END_IF
		
IF (strcmp(token, 'token_type')) THEN
	getEnumTypeFromToken := cEnumTypeTokenType;
	RETURN;
END_IF

IF (strcmp(token, 'UI_event_code')) THEN
	getEnumTypeFromToken := cEnumTypeUiEventCode;
	RETURN;
END_IF
		
IF (strcmp(token, 'ui_orientation')) THEN
	getEnumTypeFromToken := cEnumTypeUiOrientation;
	RETURN;
END_IF

parseOK := FALSE;
getEnumTypeFromToken := default;
          
END_FUNCTION

FUNCTION getProgMovCodeFromToken : t_prog_mov_code
  VAR_INPUT
    token : t_token_string;
    default : t_prog_mov_code;
    parseOK : REFERENCE TO BOOL;
  END_VAR

            IF (strcmp(token,'pmlTop')) THEN
	getProgMovCodeFromToken := cProgMovCode_Lift_Top;
	RETURN;
END_IF

IF (strcmp(token,'pmlBottom')) THEN
	getProgMovCodeFromToken := cProgMovCode_Lift_Bottom;
	RETURN;
END_IF

IF (strcmp(token,'pmlStdOnGnd')) THEN
	getProgMovCodeFromToken := cProgMovCode_Lift_StandardOnGround;
	RETURN;
END_IF

IF (strcmp(token,'pmlStdGnd')) THEN
	getProgMovCodeFromToken := cProgMovCode_Lift_StandardGround;
	RETURN;
END_IF

IF (strcmp(token,'pmlStdTruck')) THEN
	getProgMovCodeFromToken := cProgMovCode_Lift_StandardTruck;
	RETURN;
END_IF

IF (strcmp(token,'pmlStdStack1')) THEN
	getProgMovCodeFromToken := cProgMovCode_Lift_StandardStack1;
	RETURN;
END_IF

IF (strcmp(token,'pmlStdStack2')) THEN
	getProgMovCodeFromToken := cProgMovCode_Lift_StandardStack2;
	RETURN;
END_IF

IF (strcmp(token,'pmlHicOnGnd')) THEN
	getProgMovCodeFromToken := cProgMovCode_Lift_HicubeOnGround;
	RETURN;
END_IF

IF (strcmp(token,'pmlHicGnd')) THEN
	getProgMovCodeFromToken := cProgMovCode_Lift_HicubeGround;
	RETURN;
END_IF

IF (strcmp(token,'pmlHicTruck')) THEN
	getProgMovCodeFromToken := cProgMovCode_Lift_HicubeTruck;
	RETURN;
END_IF

IF (strcmp(token,'pmlHicStack1')) THEN
	getProgMovCodeFromToken := cProgMovCode_Lift_HicubeStack1;
	RETURN;
END_IF

IF (strcmp(token,'pmlHicStack2')) THEN
	getProgMovCodeFromToken := cProgMovCode_Lift_HicubeStack2;
	RETURN;
END_IF

IF (strcmp(token,'pmtLat0Fwd')) THEN
	getProgMovCodeFromToken := cProgMovCode_Travel_LAT0_Forward;
	RETURN;
END_IF

IF (strcmp(token,'pmtLat0Rev')) THEN
	getProgMovCodeFromToken := cProgMovCode_Travel_LAT0_Reverse;
	RETURN;
END_IF

IF (strcmp(token,'pmtLat04WSFwd')) THEN
	getProgMovCodeFromToken := cProgMovCode_Travel_LAT0_4WS_Forward;
	RETURN;
END_IF

IF (strcmp(token,'pmtLat04WSRev')) THEN
	getProgMovCodeFromToken := cProgMovCode_Travel_LAT0_4WS_Reverse;
	RETURN;
END_IF

IF (strcmp(token,'pmtLatPos90Fwd')) THEN
	getProgMovCodeFromToken := cProgMovCode_Travel_LATPos90_Forward;
	RETURN;
END_IF

IF (strcmp(token,'pmtLatPos90Rev')) THEN
	getProgMovCodeFromToken := cProgMovCode_Travel_LATPos90_Reverse;
	RETURN;
END_IF

IF (strcmp(token,'pmtLatNeg90Fwd')) THEN
	getProgMovCodeFromToken := cProgMovCode_Travel_LATNeg90_Forward;
	RETURN;
END_IF

IF (strcmp(token,'pmtLatNeg90Rev')) THEN
	getProgMovCodeFromToken := cProgMovCode_Travel_LATNeg90_Reverse;
	RETURN;
END_IF

IF (strcmp(token,'pmTest1')) THEN
	getProgMovCodeFromToken := cProgMovCode_Test1;
	RETURN;
END_IF

IF (strcmp(token,'pmTest2')) THEN
	getProgMovCodeFromToken := cProgMovCode_Test2;
	RETURN;
END_IF

IF (strcmp(token,'pms0')) THEN
	getProgMovCodeFromToken := cProgMovCode_Steer_0;
	RETURN;
END_IF

IF (strcmp(token,'pmClear')) THEN
	getProgMovCodeFromToken := cProgMovCode_Clear;
	RETURN;
END_IF

IF (strcmp(token,'none')) THEN
	getProgMovCodeFromToken := cProgMovCodeNone;
	RETURN;
END_IF

parseOK := FALSE;
getProgMovCodeFromToken := default;

          
END_FUNCTION

FUNCTION getStringForEnumOptions : STRING
  VAR_INPUT
    enum : t_enum_type;
  END_VAR

            getStringForEnumOptions := '["ab", "bc", "cd", "ef"]';

(*
CASE enum OF
	cEnumTypeNone:
		getStringForEnumType := 'int';
	
	cEnumTypeActiveState:
		getStringForEnumType := 'active_state';
		
	cEnumTypeBMSChargeState:
		getStringForEnumType := 'BMS_charge_state';

	cEnumTypeBMSFaultLevel:
		getStringForEnumType := 'BMS_fault_level';
		
	cEnumTypeBMSState:
		getStringForEnumType := 'BMS_state';
		
	cEnumTypeChannelMask:
		getStringForEnumType := 'channel_mask';
		
	cEnumTypeChargeQualifier:
		getStringForEnumType := 'charge_qualifier';

	cEnumTypeDebugMask:
		getStringForEnumType := 'debug_mask';
		
	cEnumTypeEventCode:
		getStringForEnumType := 'event_code';

	cEnumTypeFunctionalMode:
		getStringForEnumType := 'functional_mode';
		
	cEnumTypeInputMode:
		getStringForEnumType := 'input_mode';
		
	cEnumTypeInterlockState:
		getStringForEnumType := 'interlock_state';

	cEnumTypeLockState:
		getStringForEnumType := 'lock_state';

	cEnumTypeOBCState:
		getStringForEnumType := 'OBC_state';
		
	cEnumTypeOBCStatus:
		getStringForEnumType := 'OBC_status';
		
	cEnumTypeOperatingMethod:
		getStringForEnumType := 'operating_method';
		
	cEnumTypeProgMovCode:
		getStringForEnumType := 'prog_mov_code';
		
	cEnumTypeRunState:
		getStringForEnumType := 'run_state';
		
	cEnumTypeSeverity:
		getStringForEnumType := 'severity';

	cEnumTypeShutdownCode:
		getStringForEnumType := 'shutdown_code';

	cEnumTypeStateCode:
		getStringForEnumType := 'state_code';

	cEnumTypeSteerMode:
		getStringForEnumType := 'steer_mode';
		
	cEnumTypeSubsystem:
		getStringForEnumType := 'subsystem';

	cEnumTypeSystemControl:
		getStringForEnumType := 'system_control';

	cEnumTypeSystemState:
		getStringForEnumType := 'system_state';
		
	cEnumTypeTMSState:
		getStringForEnumType := 'TMS_state';
		
	cEnumTypeTokenType:
		getStringForEnumType := 'token_type';

	cEnumTypeUiEventCode:
		getStringForEnumType := 'UI_event_code';
		
	cEnumTypeUiOrientation:
		getStringForEnumType := 'ui_orientation';
END_CASE
*)
          
END_FUNCTION

FUNCTION getStringForProgMovCode : t_medium_string
  VAR_INPUT
    state : t_prog_mov_code;
  END_VAR

            getStringForProgMovCode := 'pmNone';

CASE state OF
	cProgMovCode_Lift_Top:
		getStringForProgMovCode := 'pmlTop';

	cProgMovCode_Lift_Bottom:
		getStringForProgMovCode := 'pmlBottom';
	
	cProgMovCode_Lift_StandardOnGround:
		getStringForProgMovCode := 'pmlStdOnGnd';

	cProgMovCode_Lift_StandardGround:
		getStringForProgMovCode := 'pmlStdGnd';

	cProgMovCode_Lift_StandardTruck:
		getStringForProgMovCode := 'pmlStdTruck';

	cProgMovCode_Lift_StandardStack1:  
		getStringForProgMovCode := 'pmlStdStack1';

	cProgMovCode_Lift_StandardStack2: 
		getStringForProgMovCode := 'pmlStdStack2';
	
	cProgMovCode_Lift_HicubeOnGround: 
		getStringForProgMovCode := 'pmlHicOnGnd';

	cProgMovCode_Lift_HicubeGround:
		getStringForProgMovCode := 'pmlHicGnd';

	cProgMovCode_Lift_HicubeTruck:
		getStringForProgMovCode := 'pmlHicTruck';

	cProgMovCode_Lift_HicubeStack1:  
		getStringForProgMovCode := 'pmlHicStack1';

	cProgMovCode_Lift_HicubeStack2: 
		getStringForProgMovCode := 'pmlHicStack2';
			
	cProgMovCode_Travel_LAT0_Forward:  
		getStringForProgMovCode := 'pmtLat0Fwd';

	cProgMovCode_Travel_LAT0_Reverse: 
		getStringForProgMovCode := 'pmtLat0Rev';

	cProgMovCode_Travel_LAT0_4WS_Forward:  
		getStringForProgMovCode := 'pmtLat04WSFwd';

	cProgMovCode_Travel_LAT0_4WS_Reverse: 
		getStringForProgMovCode := 'pmtLat04WSRev';
	
	cProgMovCode_Travel_LATPos90_Forward: 
		getStringForProgMovCode := 'pmtLatPos90Fwd';

	cProgMovCode_Travel_LATPos90_Reverse: 
		getStringForProgMovCode := 'pmtLatPos90Rev';

	cProgMovCode_Travel_LATNeg90_Forward: 
		getStringForProgMovCode := 'pmtLatNeg90Fwd';

	cProgMovCode_Travel_LATNeg90_Reverse: 
		getStringForProgMovCode := 'pmtLatNeg90Rev';
	
	cProgMovCode_Test1:
		getStringForProgMovCode := 'pmTest1';

	cProgMovCode_Test2: 
		getStringForProgMovCode := 'pmTest2';

	cProgMovCode_Steer_0:  
		getStringForProgMovCode := 'pms0';

	cProgMovCode_Clear:
		getStringForProgMovCode := 'pmClear';
END_CASE

          
END_FUNCTION

FUNCTION getStringForSeverity : t_medium_string
  VAR_INPUT
    severity : t_severity;
  END_VAR

            getStringForSeverity := 'none';

CASE severity OF
	cSeverityWarning: 
		getStringForSeverity := 'warning';
	
	cSeverityError:
		getStringForSeverity := 'error';
	
	cSeverityCritical:
		getStringForSeverity := 'critical';	
END_CASE
          
END_FUNCTION

FUNCTION getStringForShutdownCode : t_medium_string
  VAR_INPUT
    code : t_shutdown_code;
  END_VAR

            getStringForShutdownCode := 'unknown';

CASE code OF
	cShutdownCodeIgnition: 
		getStringForShutdownCode := 'ignition';
	
	cShutdownCodeSoftware:
		getStringForShutdownCode := 'software';
	
	cShutdownCodeSupervisor:
		getStringForShutdownCode := 'supervisor';	
	
	cShutdownCodeCrashDetected:
		getStringForShutdownCode := 'crash';	
	
	cShutdownCodeTrapDetected:
		getStringForShutdownCode := 'trap';
END_CASE

          
END_FUNCTION

FUNCTION getStringForSystemControl : t_medium_string
  VAR_INPUT
    control : t_system_control;
  END_VAR

            getStringForSystemControl := 'unknown';

CASE control OF
	cSystemControlEStop:
		getStringForSystemControl := 'estop';

	cSystemControlReset:
		getStringForSystemControl := 'reset';

	cSystemControlStop:
		getStringForSystemControl := 'stop';
		
	cSystemControlStart:
		getStringForSystemControl := 'start';

	cSystemControlNone:
		getStringForSystemControl := 'none';	
END_CASE
          
END_FUNCTION

FUNCTION getStringForTokenType : t_medium_string
  VAR_INPUT
    token : t_token_type;
  END_VAR

            getStringForTokenType := 'none';

CASE token OF
	cTokenDescribe:
		getStringForTokenType := 'describe';
		
	cTokenSyntax:
		getStringForTokenType := 'syntax';
			
	cTokenVerify:
		getStringForTokenType := 'verify';
			
	cTokenIdentify:
		getStringForTokenType := 'identity';
			
	cTokenRegister:
		getStringForTokenType := 'register';
			
	cTokenConfigure:
		getStringForTokenType := 'configure';
		
	cTokenSetFailSafeMode:
		getStringForTokenType := 'failsafe_set';
			
	cTokenClearFailSafeMode:
		getStringForTokenType := 'failsafe_clear';
			
	cTokenFailSafeConfig:
		getStringForTokenType := 'failsafe_config';
			
	cTokenProceed:
		getStringForTokenType := 'proceed';
			
	cTokenDebugMaskAdd:
		getStringForTokenType := 'debug_add';
			
	cTokenDebugMaskDelete:
		getStringForTokenType := 'debug_del';
			
	cTokenDebugMaskClear:
		getStringForTokenType := 'debug_clear';
			
	cTokenClose:
		getStringForTokenType := 'close';
			
	cTokenExport:
		getStringForTokenType := 'export';
			
	cTokenClear:
		getStringForTokenType := 'clear';
			
	cTokenDeregister:
		getStringForTokenType := 'deregister';
			
	cTokenTrigger:
		getStringForTokenType := 'trigger';
			
	cTokenChannelMaskAdd:
		getStringForTokenType := 'chan_add';
			
	cTokenChannelMaskDelete:
		getStringForTokenType := 'chan_del';
			
	cTokenChannelMaskClear:
		getStringForTokenType := 'chan_clear';
			
	cTokenChannelIndex:
		getStringForTokenType := '<index>';
END_CASE

	

//	: t_medium_string:= 'value_type';
//	: t_medium_string:= 'meaning';
          
END_FUNCTION

FUNCTION getTokenTypeFromToken : t_token_type
  VAR_INPUT
    token : t_token_string;
    default : t_token_type;
    parseOK : REFERENCE TO BOOL;
  END_VAR

            parseOK := FALSE;
getTokenTypeFromToken := default;


          
END_FUNCTION

FUNCTION splitFQN : BOOL
  VAR_INPUT
    fqn : REFERENCE TO t_fqtoken_string;
    tokens : REFERENCE TO t_token_string_set;
    count : REFERENCE TO USINT;
  END_VAR
  VAR
    i : USINT;
    position : USINT;
    length : USINT;
    currentLength : USINT;
  END_VAR

            length := INT_TO_USINT(len(fqn));

count := 0;
position := 1;
currentLength := 0;

FOR i:=1 TO length DO
	IF (fqn[i-1]=46) THEN
		IF (count>=cTokenStringSetCount) THEN
			splitFQN := FALSE;
			RETURN;
		END_IF
		
		count := count + 1;
		tokens[count] := MID(fqn,currentLength,position);
		
		currentLength := 0;
		position := i + 1;
	ELSE
		currentLength := currentLength + 1;
		IF (currentLength>INT_TO_USINT(SIZEOF(t_token_string)-1)) THEN
			splitFQN := FALSE;
			RETURN;
		END_IF
	END_IF
END_FOR

IF (currentLength=0) THEN
	RETURN;
END_IF

